gfCNCPoint6[8476] = {X 389.8299, Y 54.3240, Z -8.0000, A 0.000, B 0.000, C 0.000 }
gfCNCPoint6[8477] = {X 390.6035, Y 54.8101, Z -8.0000, A 0.000, B 0.000, C 0.000 }
gfCNCPoint6[8478] = {X 391.2496, Y 55.4562, Z -8.0000, A 0.000, B 0.000, C 0.000 }
gfCNCPoint6[8479] = {X 391.7356, Y 56.2298, Z -8.0000, A 0.000, B 0.000, C 0.000 }
gfCNCPoint6[8480] = {X 392.0374, Y 57.0921, Z -8.0000, A 0.000, B 0.000, C 0.000 }
gfCNCPoint6[8481] = {X 392.1397, Y 58.0000, Z -8.0000, A 0.000, B 0.000, C 0.000 }
gfCNCPoint6[8482] = {X 392.1397, Y 58.9342, Z -8.0000, A 0.000, B 0.000, C 0.000 }
gfCNCPoint6[8483] = {X 392.0387, Y 59.8361, Z -8.0000, A 0.000, B 0.000, C 0.000 }
gfCNCPoint6[8484] = {X 391.7409, Y 60.6934, Z -8.0000, A 0.000, B 0.000, C 0.000 }
gfCNCPoint6[8485] = {X 391.2105, Y 61.5272, Z -8.0000, A 0.000, B 0.000, C 0.000 }
gfCNCPoint6[8486] = {X 390.4961, Y 62.2101, Z -8.0000, A 0.000, B 0.000, C 0.000 }
gfCNCPoint6[8487] = {X 389.6392, Y 62.7024, Z -8.0000, A 0.000, B 0.000, C 0.000 }
gfCNCPoint6[8488] = {X 388.6895, Y 62.9755, Z -8.0000, A 0.000, B 0.000, C 0.000 }
gfCNCPoint6[8489] = {X 388.5563, Y 62.9947, Z -8.0000, A 0.000, B 0.000, C 0.000 }
gfCNCPoint6[8490] = {X 388.4224, Y 63.0095, Z -8.0000, A 0.000, B 0.000, C 0.000 }
gfCNCPoint6[8491] = {X 388.4203, Y 63.1546, Z -8.0000, A 0.000, B 0.000, C 0.000 }
gfCNCPoint6[8492] = {X 388.4183, Y 84.6157, Z -8.0000, A 0.000, B 0.000, C 0.000 }
gfCNCPoint6[8493] = {X 388.3592, Y 86.2534, Z -8.0000, A 0.000, B 0.000, C 0.000 }
gfCNCPoint6[8494] = {X 388.1574, Y 87.8797, Z -8.0000, A 0.000, B 0.000, C 0.000 }
gfCNCPoint6[8495] = {X 387.8145, Y 89.4823, Z -8.0000, A 0.000, B 0.000, C 0.000 }
gfCNCPoint6[8496] = {X 387.2961, Y 91.0293, Z -8.0000, A 0.000, B 0.000, C 0.000 }
gfCNCPoint6[8497] = {X 386.5671, Y 92.4889, Z -8.0000, A 0.000, B 0.000, C 0.000 }
gfCNCPoint6[8498] = {X 385.6417, Y 93.8327, Z -8.0000, A 0.000, B 0.000, C 0.000 }
gfCNCPoint6[8499] = {X 384.5380, Y 95.0343, Z -8.0000, A 0.000, B 0.000, C 0.000 }
gfCNCPoint6[8500] = {X 383.0366, Y 96.3053, Z -8.0000, A 0.000, B 0.000, C 0.000 }
gfCNCPoint6[8501] = {X 381.4074, Y 97.4078, Z -8.0000, A 0.000, B 0.000, C 0.000 }
gfCNCPoint6[8502] = {X 379.6693, Y 98.3292, Z -8.0000, A 0.000, B 0.000, C 0.000 }
gfCNCPoint6[8503] = {X 377.4136, Y 99.2775, Z -8.0000, A 0.000, B 0.000, C 0.000 }
gfCNCPoint6[8504] = {X 375.0960, Y 100.0622, Z -8.0000, A 0.000, B 0.000, C 0.000 }
gfCNCPoint6[8505] = {X 372.7282, Y 100.6793, Z -8.0000, A 0.000, B 0.000, C 0.000 }
gfCNCPoint6[8506] = {X 369.0580, Y 101.3935, Z -8.0000, A 0.000, B 0.000, C 0.000 }
gfCNCPoint6[8507] = {X 365.3582, Y 101.9340, Z -8.0000, A 0.000, B 0.000, C 0.000 }
gfCNCPoint6[8508] = {X 361.6370, Y 102.2996, Z -8.0000, A 0.000, B 0.000, C 0.000 }
gfCNCPoint6[8509] = {X 355.6353, Y 102.6431, Z -8.0000, A 0.000, B 0.000, C 0.000 }
gfCNCPoint6[8510] = {X 349.6255, Y 102.7879, Z -8.0000, A 0.000, B 0.000, C 0.000 }
gfCNCPoint6[8511] = {X 349.6557, Y 106.7878, Z -8.0000, A 0.000, B 0.000, C 0.000 }
gfCNCPoint6[8512] = {X 349.6556, Y 106.7878, Z -8.0000, A 0.000, B 0.000, C 0.000 }
gfCNCPoint6[8513] = {X 349.6249, Y 102.7077, Z -8.0000, A 0.000, B 0.000, C 0.000 }
gfCNCPoint6[8514] = {X 346.2791, Y 102.7021, Z -8.0000, A 0.000, B 0.000, C 0.000 }
gfCNCPoint6[8515] = {X 342.9340, Y 102.6349, Z -8.0000, A 0.000, B 0.000, C 0.000 }
gfCNCPoint6[8516] = {X 342.4013, Y 102.6162, Z -8.0000, A 0.000, B 0.000, C 0.000 }
gfCNCPoint6[8517] = {X 342.2415, Y 102.6136, Z -8.0000, A 0.000, B 0.000, C 0.000 }
gfCNCPoint6[8518] = {X 337.6107, Y 102.4240, Z -8.0000, A 0.000, B 0.000, C 0.000 }
gfCNCPoint6[8519] = {X 332.9916, Y 102.0451, Z -8.0000, A 0.000, B 0.000, C 0.000 }
gfCNCPoint6[8520] = {X 328.3918, Y 101.4774, Z -8.0000, A 0.000, B 0.000, C 0.000 }
gfCNCPoint6[8521] = {X 325.3437, Y 100.9426, Z -8.0000, A 0.000, B 0.000, C 0.000 }
gfCNCPoint6[8522] = {X 322.3384, Y 100.2041, Z -8.0000, A 0.000, B 0.000, C 0.000 }
gfCNCPoint6[8523] = {X 319.3896, Y 99.2654, Z -8.0000, A 0.000, B 0.000, C 0.000 }
gfCNCPoint6[8524] = {X 317.6756, Y 98.5798, Z -8.0000, A 0.000, B 0.000, C 0.000 }
gfCNCPoint6[8525] = {X 316.0258, Y 97.7518, Z -8.0000, A 0.000, B 0.000, C 0.000 }
gfCNCPoint6[8526] = {X 314.4519, Y 96.7872, Z -8.0000, A 0.000, B 0.000, C 0.000 }
gfCNCPoint6[8527] = {X 312.9652, Y 95.6930, Z -8.0000, A 0.000, B 0.000, C 0.000 }
gfCNCPoint6[8528] = {X 311.8398, Y 94.6644, Z -8.0000, A 0.000, B 0.000, C 0.000 }
gfCNCPoint6[8529] = {X 310.8546, Y 93.5009, Z -8.0000, A 0.000, B 0.000, C 0.000 }
gfCNCPoint6[8530] = {X 310.0255, Y 92.2214, Z -8.0000, A 0.000, B 0.000, C 0.000 }
gfCNCPoint6[8531] = {X 309.3660, Y 90.8468, Z -8.0000, A 0.000, B 0.000, C 0.000 }
gfCNCPoint6[8532] = {X 308.8111, Y 89.0438, Z -8.0000, A 0.000, B 0.000, C 0.000 }
gfCNCPoint6[8533] = {X 308.4634, Y 87.1897, Z -8.0000, A 0.000, B 0.000, C 0.000 }
gfCNCPoint6[8534] = {X 308.3276, Y 85.3082, Z -8.0000, A 0.000, B 0.000, C 0.000 }
gfCNCPoint6[8535] = {X 308.3140, Y 84.6159, Z -8.0000, A 0.000, B 0.000, C 0.000 }
gfCNCPoint6[8536] = {X 308.3153, Y 62.9242, Z -8.0000, A 0.000, B 0.000, C 0.000 }
gfCNCPoint6[8537] = {X 307.4730, Y 62.7731, Z -8.0000, A 0.000, B 0.000, C 0.000 }
gfCNCPoint6[8538] = {X 306.6820, Y 62.4463, Z -8.0000, A 0.000, B 0.000, C 0.000 }
gfCNCPoint6[8539] = {X 305.9787, Y 61.9587, Z -8.0000, A 0.000, B 0.000, C 0.000 }
gfCNCPoint6[8540] = {X 305.3952, Y 61.3327, Z -8.0000, A 0.000, B 0.000, C 0.000 }
gfCNCPoint6[8541] = {X 304.9582, Y 60.5969, Z -8.0000, A 0.000, B 0.000, C 0.000 }
gfCNCPoint6[8542] = {X 304.6878, Y 59.7849, Z -8.0000, A 0.000, B 0.000, C 0.000 }
gfCNCPoint6[8543] = {X 304.5962, Y 58.9341, Z -8.0000, A 0.000, B 0.000, C 0.000 }
gfCNCPoint6[8544] = {X 304.5962, Y 58.0000, Z -8.0000, A 0.000, B 0.000, C 0.000 }
gfCNCPoint6[8545] = {X 304.6965, Y 57.1099, Z -8.0000, A 0.000, B 0.000, C 0.000 }
gfCNCPoint6[8546] = {X 304.9923, Y 56.2645, Z -8.0000, A 0.000, B 0.000, C 0.000 }
gfCNCPoint6[8547] = {X 305.4689, Y 55.5060, Z -8.0000, A 0.000, B 0.000, C 0.000 }
gfCNCPoint6[8548] = {X 306.1023, Y 54.8727, Z -8.0000, A 0.000, B 0.000, C 0.000 }
gfCNCPoint6[8549] = {X 306.8607, Y 54.3961, Z -8.0000, A 0.000, B 0.000, C 0.000 }
gfCNCPoint6[8550] = {X 307.7061, Y 54.1003, Z -8.0000, A 0.000, B 0.000, C 0.000 }
gfCNCPoint6[8551] = {X 308.5962, Y 54.0000, Z -8.0000, A 0.000, B 0.000, C 0.000 }
gfCNCPoint6[8552] = {X 324.3107, Y 54.0000, Z -8.0000, A 0.000, B 0.000, C 0.000 }
gfCNCPoint6[8553] = {X 325.2008, Y 54.1003, Z -8.0000, A 0.000, B 0.000, C 0.000 }
gfCNCPoint6[8554] = {X 326.0462, Y 54.3961, Z -8.0000, A 0.000, B 0.000, C 0.000 }
gfCNCPoint6[8555] = {X 326.8046, Y 54.8727, Z -8.0000, A 0.000, B 0.000, C 0.000 }
gfCNCPoint6[8556] = {X 327.4380, Y 55.5060, Z -8.0000, A 0.000, B 0.000, C 0.000 }
gfCNCPoint6[8557] = {X 327.9146, Y 56.2645, Z -8.0000, A 0.000, B 0.000, C 0.000 }
gfCNCPoint6[8558] = {X 328.2104, Y 57.1099, Z -8.0000, A 0.000, B 0.000, C 0.000 }
gfCNCPoint6[8559] = {X 328.3107, Y 58.0000, Z -8.0000, A 0.000, B 0.000, C 0.000 }
gfCNCPoint6[8560] = {X 328.3107, Y 58.9341, Z -8.0000, A 0.000, B 0.000, C 0.000 }
gfCNCPoint6[8561] = {X 328.2156, Y 59.7845, Z -8.0000, A 0.000, B 0.000, C 0.000 }
gfCNCPoint6[8562] = {X 327.9434, Y 60.5958, Z -8.0000, A 0.000, B 0.000, C 0.000 }
gfCNCPoint6[8563] = {X 327.5064, Y 61.3315, Z -8.0000, A 0.000, B 0.000, C 0.000 }
gfCNCPoint6[8564] = {X 326.9240, Y 61.9586, Z -8.0000, A 0.000, B 0.000, C 0.000 }
gfCNCPoint6[8565] = {X 326.2226, Y 62.4488, Z -8.0000, A 0.000, B 0.000, C 0.000 }
gfCNCPoint6[8566] = {X 325.4337, Y 62.7801, Z -8.0000, A 0.000, B 0.000, C 0.000 }
gfCNCPoint6[8567] = {X 324.5926, Y 62.9377, Z -8.0000, A 0.000, B 0.000, C 0.000 }
gfCNCPoint6[8568] = {X 324.5946, Y 83.2313, Z -8.0000, A 0.000, B 0.000, C 0.000 }
gfCNCPoint6[8569] = {X 324.6081, Y 84.6159, Z -8.0000, A 0.000, B 0.000, C 0.000 }
gfCNCPoint6[8570] = {X 324.6916, Y 85.9176, Z -8.0000, A 0.000, B 0.000, C 0.000 }
gfCNCPoint6[8571] = {X 324.9294, Y 87.2002, Z -8.0000, A 0.000, B 0.000, C 0.000 }
gfCNCPoint6[8572] = {X 325.4490, Y 87.7103, Z -8.0000, A 0.000, B 0.000, C 0.000 }
gfCNCPoint6[8573] = {X 326.0776, Y 88.0775, Z -8.0000, A 0.000, B 0.000, C 0.000 }
gfCNCPoint6[8574] = {X 327.8904, Y 88.8015, Z -8.0000, A 0.000, B 0.000, C 0.000 }
gfCNCPoint6[8575] = {X 329.7768, Y 89.3033, Z -8.0000, A 0.000, B 0.000, C 0.000 }
gfCNCPoint6[8576] = {X 332.8789, Y 89.8598, Z -8.0000, A 0.000, B 0.000, C 0.000 }
gfCNCPoint6[8577] = {X 336.0092, Y 90.2262, Z -8.0000, A 0.000, B 0.000, C 0.000 }
gfCNCPoint6[8578] = {X 340.3892, Y 90.5211, Z -8.0000, A 0.000, B 0.000, C 0.000 }
gfCNCPoint6[8579] = {X 344.7764, Y 90.6753, Z -8.0000, A 0.000, B 0.000, C 0.000 }
gfCNCPoint6[8580] = {X 349.1664, Y 90.6886, Z -8.0000, A 0.000, B 0.000, C 0.000 }
gfCNCPoint6[8581] = {X 353.3283, Y 90.6201, Z -8.0000, A 0.000, B 0.000, C 0.000 }
gfCNCPoint6[8582] = {X 357.4851, Y 90.4005, Z -8.0000, A 0.000, B 0.000, C 0.000 }
gfCNCPoint6[8583] = {X 361.6311, Y 90.0301, Z -8.0000, A 0.000, B 0.000, C 0.000 }
gfCNCPoint6[8584] = {X 363.7299, Y 89.7406, Z -8.0000, A 0.000, B 0.000, C 0.000 }
gfCNCPoint6[8585] = {X 365.8095, Y 89.3352, Z -8.0000, A 0.000, B 0.000, C 0.000 }
gfCNCPoint6[8586] = {X 367.8634, Y 88.8152, Z -8.0000, A 0.000, B 0.000, C 0.000 }
gfCNCPoint6[8587] = {X 368.8291, Y 88.4908, Z -8.0000, A 0.000, B 0.000, C 0.000 }
gfCNCPoint6[8588] = {X 369.7521, Y 88.0599, Z -8.0000, A 0.000, B 0.000, C 0.000 }
gfCNCPoint6[8589] = {X 370.6208, Y 87.5278, Z -8.0000, A 0.000, B 0.000, C 0.000 }
gfCNCPoint6[8590] = {X 370.8574, Y 87.2814, Z -8.0000, A 0.000, B 0.000, C 0.000 }
gfCNCPoint6[8591] = {X 370.9793, Y 86.9624, Z -8.0000, A 0.000, B 0.000, C 0.000 }
gfCNCPoint6[8592] = {X 371.1738, Y 85.4011, Z -8.0000, A 0.000, B 0.000, C 0.000 }
gfCNCPoint6[8593] = {X 371.2387, Y 83.8290, Z -8.0000, A 0.000, B 0.000, C 0.000 }
gfCNCPoint6[8594] = {X 371.2376, Y 63.0401, Z -8.0000, A 0.000, B 0.000, C 0.000 }
gfCNCPoint6[8595] = {X 371.2440, Y 62.9246, Z -8.0000, A 0.000, B 0.000, C 0.000 }
gfCNCPoint6[8596] = {X 371.0714, Y 62.9089, Z -8.0000, A 0.000, B 0.000, C 0.000 }
gfCNCPoint6[8597] = {X 370.8996, Y 62.8858, Z -8.0000, A 0.000, B 0.000, C 0.000 }
gfCNCPoint6[8598] = {X 369.9933, Y 62.6315, Z -8.0000, A 0.000, B 0.000, C 0.000 }
gfCNCPoint6[8599] = {X 369.1714, Y 62.1725, Z -8.0000, A 0.000, B 0.000, C 0.000 }
gfCNCPoint6[8600] = {X 368.4796, Y 61.5342, Z -8.0000, A 0.000, B 0.000, C 0.000 }
gfCNCPoint6[8601] = {X 367.9562, Y 60.7518, Z -8.0000, A 0.000, B 0.000, C 0.000 }
gfCNCPoint6[8602] = {X 367.6300, Y 59.8688, Z -8.0000, A 0.000, B 0.000, C 0.000 }
gfCNCPoint6[8603] = {X 367.5193, Y 58.9341, Z -8.0000, A 0.000, B 0.000, C 0.000 }
gfCNCPoint6[8604] = {X 367.5193, Y 58.0000, Z -8.0000, A 0.000, B 0.000, C 0.000 }
gfCNCPoint6[8605] = {X 367.6196, Y 57.1099, Z -8.0000, A 0.000, B 0.000, C 0.000 }
gfCNCPoint6[8606] = {X 367.9154, Y 56.2645, Z -8.0000, A 0.000, B 0.000, C 0.000 }
gfCNCPoint6[8607] = {X 368.3920, Y 55.5060, Z -8.0000, A 0.000, B 0.000, C 0.000 }
gfCNCPoint6[8608] = {X 369.0253, Y 54.8727, Z -8.0000, A 0.000, B 0.000, C 0.000 }
gfCNCPoint6[8609] = {X 369.7837, Y 54.3961, Z -8.0000, A 0.000, B 0.000, C 0.000 }
gfCNCPoint6[8610] = {X 370.6292, Y 54.1003, Z -8.0000, A 0.000, B 0.000, C 0.000 }
gfCNCPoint6[8611] = {X 371.5193, Y 54.0000, Z -8.0000, A 0.000, B 0.000, C 0.000 }
gfCNCPoint6[8612] = {X 388.0597, Y 54.0000, Z -8.0000, A 0.000, B 0.000, C 0.000 }
gfCNCPoint6[8613] = {X 388.9498, Y 54.1003, Z -8.0000, A 0.000, B 0.000, C 0.000 }
gfCNCPoint6[8614] = {X 389.7952, Y 54.3961, Z -8.0000, A 0.000, B 0.000, C 0.000 }
gfCNCPoint6[8615] = {X 390.5536, Y 54.8727, Z -8.0000, A 0.000, B 0.000, C 0.000 }
gfCNCPoint6[8616] = {X 391.1870, Y 55.5060, Z -8.0000, A 0.000, B 0.000, C 0.000 }
gfCNCPoint6[8617] = {X 391.6636, Y 56.2645, Z -8.0000, A 0.000, B 0.000, C 0.000 }
gfCNCPoint6[8618] = {X 391.9594, Y 57.1099, Z -8.0000, A 0.000, B 0.000, C 0.000 }
gfCNCPoint6[8619] = {X 392.0597, Y 58.0000, Z -8.0000, A 0.000, B 0.000, C 0.000 }
gfCNCPoint6[8620] = {X 392.0595, Y 58.9671, Z -8.0000, A 0.000, B 0.000, C 0.000 }
gfCNCPoint6[8621] = {X 391.9570, Y 59.8345, Z -8.0000, A 0.000, B 0.000, C 0.000 }
gfCNCPoint6[8622] = {X 391.6687, Y 60.6589, Z -8.0000, A 0.000, B 0.000, C 0.000 }
gfCNCPoint6[8623] = {X 391.1486, Y 61.4765, Z -8.0000, A 0.000, B 0.000, C 0.000 }
gfCNCPoint6[8624] = {X 390.4482, Y 62.1460, Z -8.0000, A 0.000, B 0.000, C 0.000 }
gfCNCPoint6[8625] = {X 389.6080, Y 62.6287, Z -8.0000, A 0.000, B 0.000, C 0.000 }
gfCNCPoint6[8626] = {X 388.6768, Y 62.8965, Z -8.0000, A 0.000, B 0.000, C 0.000 }
gfCNCPoint6[8627] = {X 388.5106, Y 62.9197, Z -8.0000, A 0.000, B 0.000, C 0.000 }
gfCNCPoint6[8628] = {X 388.3435, Y 62.9359, Z -8.0000, A 0.000, B 0.000, C 0.000 }
gfCNCPoint6[8629] = {X 388.3403, Y 63.1540, Z -8.0000, A 0.000, B 0.000, C 0.000 }
gfCNCPoint6[8630] = {X 388.3403, Y 83.9236, Z -8.0000, A 0.000, B 0.000, C 0.000 }
gfCNCPoint6[8631] = {X 388.3383, Y 84.6159, Z -8.0000, A 0.000, B 0.000, C 0.000 }
gfCNCPoint6[8632] = {X 388.2794, Y 86.2468, Z -8.0000, A 0.000, B 0.000, C 0.000 }
gfCNCPoint6[8633] = {X 388.0785, Y 87.8663, Z -8.0000, A 0.000, B 0.000, C 0.000 }
gfCNCPoint6[8634] = {X 387.7371, Y 89.4621, Z -8.0000, A 0.000, B 0.000, C 0.000 }
gfCNCPoint6[8635] = {X 387.2222, Y 90.9986, Z -8.0000, A 0.000, B 0.000, C 0.000 }
gfCNCPoint6[8636] = {X 386.4982, Y 92.4482, Z -8.0000, A 0.000, B 0.000, C 0.000 }
gfCNCPoint6[8637] = {X 385.5792, Y 93.7828, Z -8.0000, A 0.000, B 0.000, C 0.000 }
gfCNCPoint6[8638] = {X 384.4830, Y 94.9762, Z -8.0000, A 0.000, B 0.000, C 0.000 }
gfCNCPoint6[8639] = {X 382.9881, Y 96.2416, Z -8.0000, A 0.000, B 0.000, C 0.000 }
gfCNCPoint6[8640] = {X 381.3661, Y 97.3393, Z -8.0000, A 0.000, B 0.000, C 0.000 }
gfCNCPoint6[8641] = {X 379.6357, Y 98.2566, Z -8.0000, A 0.000, B 0.000, C 0.000 }
gfCNCPoint6[8642] = {X 377.3853, Y 99.2027, Z -8.0000, A 0.000, B 0.000, C 0.000 }
gfCNCPoint6[8643] = {X 375.0731, Y 99.9856, Z -8.0000, A 0.000, B 0.000, C 0.000 }
gfCNCPoint6[8644] = {X 372.7108, Y 100.6012, Z -8.0000, A 0.000, B 0.000, C 0.000 }
gfCNCPoint6[8645] = {X 369.0444, Y 101.3146, Z -8.0000, A 0.000, B 0.000, C 0.000 }
gfCNCPoint6[8646] = {X 365.3484, Y 101.8546, Z -8.0000, A 0.000, B 0.000, C 0.000 }
gfCNCPoint6[8647] = {X 361.6311, Y 102.2198, Z -8.0000, A 0.000, B 0.000, C 0.000 }
gfCNCPoint6[8648] = {X 355.6320, Y 102.5630, Z -8.0000, A 0.000, B 0.000, C 0.000 }
gfCNCPoint6[8649] = {X 349.6249, Y 102.7077, Z -8.0000, A 0.000, B 0.000, C 0.000 }
gfCNCPoint6[8650] = {X 349.6556, Y 106.7878, Z -8.0000, A 0.000, B 0.000, C 0.000 }
gfCNCPoint6[8651] = {X 349.6556, Y 106.7878, Z -5.0000, A 0.000, B 0.000, C 0.000 }
gfCNCPoint6[8652] = {X 349.6556, Y 106.7878, Z 11.0000, A 0.000, B 0.000, C 0.000 }
gfCNCPoint6[8653] = {X 411.5981, Y 79.5921, Z 11.0000, A 0.000, B 0.000, C 0.000 }
gfCNCPoint6[8654] = {X 411.5981, Y 79.5921, Z -5.0000, A 0.000, B 0.000, C 0.000 }
gfCNCPoint6[8655] = {X 411.5981, Y 79.5921, Z -8.0000, A 0.000, B 0.000, C 0.000 }
gfCNCPoint6[8656] = {X 413.7984, Y 83.0280, Z -8.0000, A 0.000, B 0.000, C 0.000 }
gfCNCPoint6[8657] = {X 428.0532, Y 73.8997, Z -8.0000, A 0.000, B 0.000, C 0.000 }
gfCNCPoint6[8658] = {X 403.7556, Y 64.3672, Z -8.0000, A 0.000, B 0.000, C 0.000 }
gfCNCPoint6[8659] = {X 402.0595, Y 63.8058, Z -8.0000, A 0.000, B 0.000, C 0.000 }
gfCNCPoint6[8660] = {X 400.3122, Y 63.4333, Z -8.0000, A 0.000, B 0.000, C 0.000 }
gfCNCPoint6[8661] = {X 398.5347, Y 63.2540, Z -8.0000, A 0.000, B 0.000, C 0.000 }
gfCNCPoint6[8662] = {X 397.5821, Y 63.1425, Z -8.0000, A 0.000, B 0.000, C 0.000 }
gfCNCPoint6[8663] = {X 396.6777, Y 62.8235, Z -8.0000, A 0.000, B 0.000, C 0.000 }
gfCNCPoint6[8664] = {X 395.8659, Y 62.3129, Z -8.0000, A 0.000, B 0.000, C 0.000 }
gfCNCPoint6[8665] = {X 395.1868, Y 61.6357, Z -8.0000, A 0.000, B 0.000, C 0.000 }
gfCNCPoint6[8666] = {X 394.6738, Y 60.8255, Z -8.0000, A 0.000, B 0.000, C 0.000 }
gfCNCPoint6[8667] = {X 394.3522, Y 59.9219, Z -8.0000, A 0.000, B 0.000, C 0.000 }
gfCNCPoint6[8668] = {X 394.2379, Y 58.9697, Z -8.0000, A 0.000, B 0.000, C 0.000 }
gfCNCPoint6[8669] = {X 394.2377, Y 58.0000, Z -8.0000, A 0.000, B 0.000, C 0.000 }
gfCNCPoint6[8670] = {X 394.3460, Y 57.0387, Z -8.0000, A 0.000, B 0.000, C 0.000 }
gfCNCPoint6[8671] = {X 394.6655, Y 56.1256, Z -8.0000, A 0.000, B 0.000, C 0.000 }
gfCNCPoint6[8672] = {X 395.1802, Y 55.3065, Z -8.0000, A 0.000, B 0.000, C 0.000 }
gfCNCPoint6[8673] = {X 395.8642, Y 54.6225, Z -8.0000, A 0.000, B 0.000, C 0.000 }
gfCNCPoint6[8674] = {X 396.6833, Y 54.1078, Z -8.0000, A 0.000, B 0.000, C 0.000 }
gfCNCPoint6[8675] = {X 397.5964, Y 53.7883, Z -8.0000, A 0.000, B 0.000, C 0.000 }
gfCNCPoint6[8676] = {X 398.5577, Y 53.6800, Z -8.0000, A 0.000, B 0.000, C 0.000 }
gfCNCPoint6[8677] = {X 419.4886, Y 53.6800, Z -8.0000, A 0.000, B 0.000, C 0.000 }
gfCNCPoint6[8678] = {X 420.4499, Y 53.7883, Z -8.0000, A 0.000, B 0.000, C 0.000 }
gfCNCPoint6[8679] = {X 421.3630, Y 54.1078, Z -8.0000, A 0.000, B 0.000, C 0.000 }
gfCNCPoint6[8680] = {X 422.1821, Y 54.6225, Z -8.0000, A 0.000, B 0.000, C 0.000 }
gfCNCPoint6[8681] = {X 422.8661, Y 55.3065, Z -8.0000, A 0.000, B 0.000, C 0.000 }
gfCNCPoint6[8682] = {X 423.3808, Y 56.1256, Z -8.0000, A 0.000, B 0.000, C 0.000 }
gfCNCPoint6[8683] = {X 423.7003, Y 57.0387, Z -8.0000, A 0.000, B 0.000, C 0.000 }
gfCNCPoint6[8684] = {X 423.8086, Y 58.0000, Z -8.0000, A 0.000, B 0.000, C 0.000 }
gfCNCPoint6[8685] = {X 423.8086, Y 58.2314, Z -8.0000, A 0.000, B 0.000, C 0.000 }
gfCNCPoint6[8686] = {X 429.6116, Y 60.4920, Z -8.0000, A 0.000, B 0.000, C 0.000 }
gfCNCPoint6[8687] = {X 457.8579, Y 71.6995, Z -8.0000, A 0.000, B 0.000, C 0.000 }
gfCNCPoint6[8688] = {X 457.8601, Y 63.2123, Z -8.0000, A 0.000, B 0.000, C 0.000 }
gfCNCPoint6[8689] = {X 457.0085, Y 63.0031, Z -8.0000, A 0.000, B 0.000, C 0.000 }
gfCNCPoint6[8690] = {X 456.2167, Y 62.6262, Z -8.0000, A 0.000, B 0.000, C 0.000 }
gfCNCPoint6[8691] = {X 455.5174, Y 62.0973, Z -8.0000, A 0.000, B 0.000, C 0.000 }
gfCNCPoint6[8692] = {X 454.9393, Y 61.4380, Z -8.0000, A 0.000, B 0.000, C 0.000 }
gfCNCPoint6[8693] = {X 454.5062, Y 60.6755, Z -8.0000, A 0.000, B 0.000, C 0.000 }
gfCNCPoint6[8694] = {X 454.2359, Y 59.8413, Z -8.0000, A 0.000, B 0.000, C 0.000 }
gfCNCPoint6[8695] = {X 454.1398, Y 58.9697, Z -8.0000, A 0.000, B 0.000, C 0.000 }
gfCNCPoint6[8696] = {X 454.1396, Y 58.0000, Z -8.0000, A 0.000, B 0.000, C 0.000 }
gfCNCPoint6[8697] = {X 454.2479, Y 57.0387, Z -8.0000, A 0.000, B 0.000, C 0.000 }
gfCNCPoint6[8698] = {X 454.5674, Y 56.1256, Z -8.0000, A 0.000, B 0.000, C 0.000 }
gfCNCPoint6[8699] = {X 455.0821, Y 55.3065, Z -8.0000, A 0.000, B 0.000, C 0.000 }
gfCNCPoint6[8700] = {X 455.7661, Y 54.6225, Z -8.0000, A 0.000, B 0.000, C 0.000 }
gfCNCPoint6[8701] = {X 456.5852, Y 54.1078, Z -8.0000, A 0.000, B 0.000, C 0.000 }
gfCNCPoint6[8702] = {X 457.4983, Y 53.7883, Z -8.0000, A 0.000, B 0.000, C 0.000 }
gfCNCPoint6[8703] = {X 458.4596, Y 53.6800, Z -8.0000, A 0.000, B 0.000, C 0.000 }
gfCNCPoint6[8704] = {X 475.0000, Y 53.6800, Z -8.0000, A 0.000, B 0.000, C 0.000 }
gfCNCPoint6[8705] = {X 475.9613, Y 53.7883, Z -8.0000, A 0.000, B 0.000, C 0.000 }
gfCNCPoint6[8706] = {X 476.8744, Y 54.1078, Z -8.0000, A 0.000, B 0.000, C 0.000 }
gfCNCPoint6[8707] = {X 477.6935, Y 54.6225, Z -8.0000, A 0.000, B 0.000, C 0.000 }
gfCNCPoint6[8708] = {X 478.3775, Y 55.3065, Z -8.0000, A 0.000, B 0.000, C 0.000 }
gfCNCPoint6[8709] = {X 478.8922, Y 56.1256, Z -8.0000, A 0.000, B 0.000, C 0.000 }
gfCNCPoint6[8710] = {X 479.2117, Y 57.0387, Z -8.0000, A 0.000, B 0.000, C 0.000 }
gfCNCPoint6[8711] = {X 479.3200, Y 58.0000, Z -8.0000, A 0.000, B 0.000, C 0.000 }
gfCNCPoint6[8712] = {X 479.3200, Y 58.9342, Z -8.0000, A 0.000, B 0.000, C 0.000 }
gfCNCPoint6[8713] = {X 479.2300, Y 59.8113, Z -8.0000, A 0.000, B 0.000, C 0.000 }
gfCNCPoint6[8714] = {X 478.9638, Y 60.6518, Z -8.0000, A 0.000, B 0.000, C 0.000 }
gfCNCPoint6[8715] = {X 478.5325, Y 61.4208, Z -8.0000, A 0.000, B 0.000, C 0.000 }
gfCNCPoint6[8716] = {X 477.9541, Y 62.0862, Z -8.0000, A 0.000, B 0.000, C 0.000 }
gfCNCPoint6[8717] = {X 477.2526, Y 62.6203, Z -8.0000, A 0.000, B 0.000, C 0.000 }
gfCNCPoint6[8718] = {X 476.4572, Y 63.0009, Z -8.0000, A 0.000, B 0.000, C 0.000 }
gfCNCPoint6[8719] = {X 475.6012, Y 63.2120, Z -8.0000, A 0.000, B 0.000, C 0.000 }
gfCNCPoint6[8720] = {X 475.6017, Y 92.7672, Z -8.0000, A 0.000, B 0.000, C 0.000 }
gfCNCPoint6[8721] = {X 475.9938, Y 92.8650, Z -8.0000, A 0.000, B 0.000, C 0.000 }
gfCNCPoint6[8722] = {X 476.3804, Y 92.9828, Z -8.0000, A 0.000, B 0.000, C 0.000 }
gfCNCPoint6[8723] = {X 477.1940, Y 93.3517, Z -8.0000, A 0.000, B 0.000, C 0.000 }
gfCNCPoint6[8724] = {X 477.9137, Y 93.8808, Z -8.0000, A 0.000, B 0.000, C 0.000 }
gfCNCPoint6[8725] = {X 478.5085, Y 94.5472, Z -8.0000, A 0.000, B 0.000, C 0.000 }
gfCNCPoint6[8726] = {X 478.9527, Y 95.3222, Z -8.0000, A 0.000, B 0.000, C 0.000 }
gfCNCPoint6[8727] = {X 479.2272, Y 96.1722, Z -8.0000, A 0.000, B 0.000, C 0.000 }
gfCNCPoint6[8728] = {X 479.3200, Y 97.0606, Z -8.0000, A 0.000, B 0.000, C 0.000 }
gfCNCPoint6[8729] = {X 479.3200, Y 98.0000, Z -8.0000, A 0.000, B 0.000, C 0.000 }
gfCNCPoint6[8730] = {X 479.2117, Y 98.9613, Z -8.0000, A 0.000, B 0.000, C 0.000 }
gfCNCPoint6[8731] = {X 478.8922, Y 99.8744, Z -8.0000, A 0.000, B 0.000, C 0.000 }
gfCNCPoint6[8732] = {X 478.3775, Y 100.6935, Z -8.0000, A 0.000, B 0.000, C 0.000 }
gfCNCPoint6[8733] = {X 477.6935, Y 101.3775, Z -8.0000, A 0.000, B 0.000, C 0.000 }
gfCNCPoint6[8734] = {X 476.8744, Y 101.8922, Z -8.0000, A 0.000, B 0.000, C 0.000 }
gfCNCPoint6[8735] = {X 475.9613, Y 102.2117, Z -8.0000, A 0.000, B 0.000, C 0.000 }
gfCNCPoint6[8736] = {X 475.0000, Y 102.3200, Z -8.0000, A 0.000, B 0.000, C 0.000 }
gfCNCPoint6[8737] = {X 458.4596, Y 102.3200, Z -8.0000, A 0.000, B 0.000, C 0.000 }
gfCNCPoint6[8738] = {X 457.4983, Y 102.2117, Z -8.0000, A 0.000, B 0.000, C 0.000 }
gfCNCPoint6[8739] = {X 456.5852, Y 101.8922, Z -8.0000, A 0.000, B 0.000, C 0.000 }
gfCNCPoint6[8740] = {X 455.7661, Y 101.3775, Z -8.0000, A 0.000, B 0.000, C 0.000 }
gfCNCPoint6[8741] = {X 455.0821, Y 100.6935, Z -8.0000, A 0.000, B 0.000, C 0.000 }
gfCNCPoint6[8742] = {X 454.5674, Y 99.8744, Z -8.0000, A 0.000, B 0.000, C 0.000 }
gfCNCPoint6[8743] = {X 454.2479, Y 98.9613, Z -8.0000, A 0.000, B 0.000, C 0.000 }
gfCNCPoint6[8744] = {X 454.1396, Y 98.0000, Z -8.0000, A 0.000, B 0.000, C 0.000 }
gfCNCPoint6[8745] = {X 454.1396, Y 97.0659, Z -8.0000, A 0.000, B 0.000, C 0.000 }
gfCNCPoint6[8746] = {X 454.2295, Y 96.1891, Z -8.0000, A 0.000, B 0.000, C 0.000 }
gfCNCPoint6[8747] = {X 454.4955, Y 95.3488, Z -8.0000, A 0.000, B 0.000, C 0.000 }
gfCNCPoint6[8748] = {X 454.9265, Y 94.5800, Z -8.0000, A 0.000, B 0.000, C 0.000 }
gfCNCPoint6[8749] = {X 455.5046, Y 93.9147, Z -8.0000, A 0.000, B 0.000, C 0.000 }
gfCNCPoint6[8750] = {X 456.2057, Y 93.3805, Z -8.0000, A 0.000, B 0.000, C 0.000 }
gfCNCPoint6[8751] = {X 457.0006, Y 92.9998, Z -8.0000, A 0.000, B 0.000, C 0.000 }
gfCNCPoint6[8752] = {X 457.8563, Y 92.7883, Z -8.0000, A 0.000, B 0.000, C 0.000 }
gfCNCPoint6[8753] = {X 457.8563, Y 85.5950, Z -8.0000, A 0.000, B 0.000, C 0.000 }
gfCNCPoint6[8754] = {X 444.8604, Y 80.5006, Z -8.0000, A 0.000, B 0.000, C 0.000 }
gfCNCPoint6[8755] = {X 420.0244, Y 96.5885, Z -8.0000, A 0.000, B 0.000, C 0.000 }
gfCNCPoint6[8756] = {X 420.0267, Y 97.0651, Z -8.0000, A 0.000, B 0.000, C 0.000 }
gfCNCPoint6[8757] = {X 420.0267, Y 98.0000, Z -8.0000, A 0.000, B 0.000, C 0.000 }
gfCNCPoint6[8758] = {X 419.9184, Y 98.9613, Z -8.0000, A 0.000, B 0.000, C 0.000 }
gfCNCPoint6[8759] = {X 419.5989, Y 99.8744, Z -8.0000, A 0.000, B 0.000, C 0.000 }
gfCNCPoint6[8760] = {X 419.0842, Y 100.6935, Z -8.0000, A 0.000, B 0.000, C 0.000 }
gfCNCPoint6[8761] = {X 418.4002, Y 101.3775, Z -8.0000, A 0.000, B 0.000, C 0.000 }
gfCNCPoint6[8762] = {X 417.5811, Y 101.8922, Z -8.0000, A 0.000, B 0.000, C 0.000 }
gfCNCPoint6[8763] = {X 416.6680, Y 102.2117, Z -8.0000, A 0.000, B 0.000, C 0.000 }
gfCNCPoint6[8764] = {X 415.7067, Y 102.3200, Z -8.0000, A 0.000, B 0.000, C 0.000 }
gfCNCPoint6[8765] = {X 396.4059, Y 102.3200, Z -8.0000, A 0.000, B 0.000, C 0.000 }
gfCNCPoint6[8766] = {X 395.4447, Y 102.2117, Z -8.0000, A 0.000, B 0.000, C 0.000 }
gfCNCPoint6[8767] = {X 394.5316, Y 101.8922, Z -8.0000, A 0.000, B 0.000, C 0.000 }
gfCNCPoint6[8768] = {X 393.7125, Y 101.3775, Z -8.0000, A 0.000, B 0.000, C 0.000 }
gfCNCPoint6[8769] = {X 393.0284, Y 100.6935, Z -8.0000, A 0.000, B 0.000, C 0.000 }
gfCNCPoint6[8770] = {X 392.5138, Y 99.8744, Z -8.0000, A 0.000, B 0.000, C 0.000 }
gfCNCPoint6[8771] = {X 392.1943, Y 98.9613, Z -8.0000, A 0.000, B 0.000, C 0.000 }
gfCNCPoint6[8772] = {X 392.0859, Y 98.0000, Z -8.0000, A 0.000, B 0.000, C 0.000 }
gfCNCPoint6[8773] = {X 392.0859, Y 97.0659, Z -8.0000, A 0.000, B 0.000, C 0.000 }
gfCNCPoint6[8774] = {X 392.1937, Y 96.1069, Z -8.0000, A 0.000, B 0.000, C 0.000 }
gfCNCPoint6[8775] = {X 392.5117, Y 95.1958, Z -8.0000, A 0.000, B 0.000, C 0.000 }
gfCNCPoint6[8776] = {X 393.0240, Y 94.3780, Z -8.0000, A 0.000, B 0.000, C 0.000 }
gfCNCPoint6[8777] = {X 393.7051, Y 93.6943, Z -8.0000, A 0.000, B 0.000, C 0.000 }
gfCNCPoint6[8778] = {X 394.5210, Y 93.1789, Z -8.0000, A 0.000, B 0.000, C 0.000 }
gfCNCPoint6[8779] = {X 395.4309, Y 92.8574, Z -8.0000, A 0.000, B 0.000, C 0.000 }
gfCNCPoint6[8780] = {X 396.3894, Y 92.7460, Z -8.0000, A 0.000, B 0.000, C 0.000 }
gfCNCPoint6[8781] = {X 397.3432, Y 92.7029, Z -8.0000, A 0.000, B 0.000, C 0.000 }
gfCNCPoint6[8782] = {X 398.2936, Y 92.6130, Z -8.0000, A 0.000, B 0.000, C 0.000 }
gfCNCPoint6[8783] = {X 398.9444, Y 92.4553, Z -8.0000, A 0.000, B 0.000, C 0.000 }
gfCNCPoint6[8784] = {X 399.5436, Y 92.1563, Z -8.0000, A 0.000, B 0.000, C 0.000 }
gfCNCPoint6[8785] = {X 413.7984, Y 83.0280, Z -8.0000, A 0.000, B 0.000, C 0.000 }
gfCNCPoint6[8786] = {X 411.6413, Y 79.6595, Z -8.0000, A 0.000, B 0.000, C 0.000 }
gfCNCPoint6[8787] = {X 413.8415, Y 83.0954, Z -8.0000, A 0.000, B 0.000, C 0.000 }
gfCNCPoint6[8788] = {X 428.2284, Y 73.8825, Z -8.0000, A 0.000, B 0.000, C 0.000 }
gfCNCPoint6[8789] = {X 403.7848, Y 64.2927, Z -8.0000, A 0.000, B 0.000, C 0.000 }
gfCNCPoint6[8790] = {X 402.0799, Y 63.7285, Z -8.0000, A 0.000, B 0.000, C 0.000 }
gfCNCPoint6[8791] = {X 400.3235, Y 63.3541, Z -8.0000, A 0.000, B 0.000, C 0.000 }
gfCNCPoint6[8792] = {X 398.5367, Y 63.1740, Z -8.0000, A 0.000, B 0.000, C 0.000 }
gfCNCPoint6[8793] = {X 397.6016, Y 63.0648, Z -8.0000, A 0.000, B 0.000, C 0.000 }
gfCNCPoint6[8794] = {X 396.7136, Y 62.7520, Z -8.0000, A 0.000, B 0.000, C 0.000 }
gfCNCPoint6[8795] = {X 395.9165, Y 62.2509, Z -8.0000, A 0.000, B 0.000, C 0.000 }
gfCNCPoint6[8796] = {X 395.2496, Y 61.5863, Z -8.0000, A 0.000, B 0.000, C 0.000 }
gfCNCPoint6[8797] = {X 394.7459, Y 60.7908, Z -8.0000, A 0.000, B 0.000, C 0.000 }
gfCNCPoint6[8798] = {X 394.4301, Y 59.9039, Z -8.0000, A 0.000, B 0.000, C 0.000 }
gfCNCPoint6[8799] = {X 394.3179, Y 58.9691, Z -8.0000, A 0.000, B 0.000, C 0.000 }
gfCNCPoint6[8800] = {X 394.3177, Y 58.0000, Z -8.0000, A 0.000, B 0.000, C 0.000 }
gfCNCPoint6[8801] = {X 394.4240, Y 57.0565, Z -8.0000, A 0.000, B 0.000, C 0.000 }
gfCNCPoint6[8802] = {X 394.7376, Y 56.1603, Z -8.0000, A 0.000, B 0.000, C 0.000 }
gfCNCPoint6[8803] = {X 395.2428, Y 55.3564, Z -8.0000, A 0.000, B 0.000, C 0.000 }
gfCNCPoint6[8804] = {X 395.9141, Y 54.6850, Z -8.0000, A 0.000, B 0.000, C 0.000 }
gfCNCPoint6[8805] = {X 396.7181, Y 54.1799, Z -8.0000, A 0.000, B 0.000, C 0.000 }
gfCNCPoint6[8806] = {X 397.6142, Y 53.8663, Z -8.0000, A 0.000, B 0.000, C 0.000 }
gfCNCPoint6[8807] = {X 398.5577, Y 53.7600, Z -8.0000, A 0.000, B 0.000, C 0.000 }
gfCNCPoint6[8808] = {X 419.4886, Y 53.7600, Z -8.0000, A 0.000, B 0.000, C 0.000 }
gfCNCPoint6[8809] = {X 420.4321, Y 53.8663, Z -8.0000, A 0.000, B 0.000, C 0.000 }
gfCNCPoint6[8810] = {X 421.3283, Y 54.1799, Z -8.0000, A 0.000, B 0.000, C 0.000 }
gfCNCPoint6[8811] = {X 422.1322, Y 54.6850, Z -8.0000, A 0.000, B 0.000, C 0.000 }
gfCNCPoint6[8812] = {X 422.8036, Y 55.3564, Z -8.0000, A 0.000, B 0.000, C 0.000 }
gfCNCPoint6[8813] = {X 423.3087, Y 56.1603, Z -8.0000, A 0.000, B 0.000, C 0.000 }
gfCNCPoint6[8814] = {X 423.6223, Y 57.0565, Z -8.0000, A 0.000, B 0.000, C 0.000 }
gfCNCPoint6[8815] = {X 423.7286, Y 58.0000, Z -8.0000, A 0.000, B 0.000, C 0.000 }
gfCNCPoint6[8816] = {X 423.7286, Y 58.2861, Z -8.0000, A 0.000, B 0.000, C 0.000 }
gfCNCPoint6[8817] = {X 429.5823, Y 60.5665, Z -8.0000, A 0.000, B 0.000, C 0.000 }
gfCNCPoint6[8818] = {X 457.9378, Y 71.8173, Z -8.0000, A 0.000, B 0.000, C 0.000 }
gfCNCPoint6[8819] = {X 457.9401, Y 63.1421, Z -8.0000, A 0.000, B 0.000, C 0.000 }
gfCNCPoint6[8820] = {X 457.0916, Y 62.9473, Z -8.0000, A 0.000, B 0.000, C 0.000 }
gfCNCPoint6[8821] = {X 456.3009, Y 62.5834, Z -8.0000, A 0.000, B 0.000, C 0.000 }
gfCNCPoint6[8822] = {X 455.6011, Y 62.0656, Z -8.0000, A 0.000, B 0.000, C 0.000 }
gfCNCPoint6[8823] = {X 455.0218, Y 61.4158, Z -8.0000, A 0.000, B 0.000, C 0.000 }
gfCNCPoint6[8824] = {X 454.5874, Y 60.6614, Z -8.0000, A 0.000, B 0.000, C 0.000 }
gfCNCPoint6[8825] = {X 454.3163, Y 59.8342, Z -8.0000, A 0.000, B 0.000, C 0.000 }
gfCNCPoint6[8826] = {X 454.2197, Y 58.9691, Z -8.0000, A 0.000, B 0.000, C 0.000 }
gfCNCPoint6[8827] = {X 454.2196, Y 58.0000, Z -8.0000, A 0.000, B 0.000, C 0.000 }
gfCNCPoint6[8828] = {X 454.3259, Y 57.0565, Z -8.0000, A 0.000, B 0.000, C 0.000 }
gfCNCPoint6[8829] = {X 454.6395, Y 56.1603, Z -8.0000, A 0.000, B 0.000, C 0.000 }
gfCNCPoint6[8830] = {X 455.1446, Y 55.3564, Z -8.0000, A 0.000, B 0.000, C 0.000 }
gfCNCPoint6[8831] = {X 455.8160, Y 54.6850, Z -8.0000, A 0.000, B 0.000, C 0.000 }
gfCNCPoint6[8832] = {X 456.6199, Y 54.1799, Z -8.0000, A 0.000, B 0.000, C 0.000 }
gfCNCPoint6[8833] = {X 457.5161, Y 53.8663, Z -8.0000, A 0.000, B 0.000, C 0.000 }
gfCNCPoint6[8834] = {X 458.4596, Y 53.7600, Z -8.0000, A 0.000, B 0.000, C 0.000 }
gfCNCPoint6[8835] = {X 475.0000, Y 53.7600, Z -8.0000, A 0.000, B 0.000, C 0.000 }
gfCNCPoint6[8836] = {X 475.9435, Y 53.8663, Z -8.0000, A 0.000, B 0.000, C 0.000 }
gfCNCPoint6[8837] = {X 476.8397, Y 54.1799, Z -8.0000, A 0.000, B 0.000, C 0.000 }
gfCNCPoint6[8838] = {X 477.6436, Y 54.6850, Z -8.0000, A 0.000, B 0.000, C 0.000 }
gfCNCPoint6[8839] = {X 478.3150, Y 55.3564, Z -8.0000, A 0.000, B 0.000, C 0.000 }
gfCNCPoint6[8840] = {X 478.8201, Y 56.1603, Z -8.0000, A 0.000, B 0.000, C 0.000 }
gfCNCPoint6[8841] = {X 479.1337, Y 57.0565, Z -8.0000, A 0.000, B 0.000, C 0.000 }
gfCNCPoint6[8842] = {X 479.2400, Y 58.0000, Z -8.0000, A 0.000, B 0.000, C 0.000 }
gfCNCPoint6[8843] = {X 479.2400, Y 58.9342, Z -8.0000, A 0.000, B 0.000, C 0.000 }
gfCNCPoint6[8844] = {X 479.1496, Y 59.8048, Z -8.0000, A 0.000, B 0.000, C 0.000 }
gfCNCPoint6[8845] = {X 478.8825, Y 60.6382, Z -8.0000, A 0.000, B 0.000, C 0.000 }
gfCNCPoint6[8846] = {X 478.4499, Y 61.3990, Z -8.0000, A 0.000, B 0.000, C 0.000 }
gfCNCPoint6[8847] = {X 477.8703, Y 62.0548, Z -8.0000, A 0.000, B 0.000, C 0.000 }
gfCNCPoint6[8848] = {X 477.1684, Y 62.5777, Z -8.0000, A 0.000, B 0.000, C 0.000 }
gfCNCPoint6[8849] = {X 476.3741, Y 62.9452, Z -8.0000, A 0.000, B 0.000, C 0.000 }
gfCNCPoint6[8850] = {X 475.5212, Y 63.1419, Z -8.0000, A 0.000, B 0.000, C 0.000 }
gfCNCPoint6[8851] = {X 475.5217, Y 92.8316, Z -8.0000, A 0.000, B 0.000, C 0.000 }
gfCNCPoint6[8852] = {X 475.9416, Y 92.9336, Z -8.0000, A 0.000, B 0.000, C 0.000 }
gfCNCPoint6[8853] = {X 476.3551, Y 93.0587, Z -8.0000, A 0.000, B 0.000, C 0.000 }
gfCNCPoint6[8854] = {X 477.1535, Y 93.4207, Z -8.0000, A 0.000, B 0.000, C 0.000 }
gfCNCPoint6[8855] = {X 477.8599, Y 93.9400, Z -8.0000, A 0.000, B 0.000, C 0.000 }
gfCNCPoint6[8856] = {X 478.4436, Y 94.5940, Z -8.0000, A 0.000, B 0.000, C 0.000 }
gfCNCPoint6[8857] = {X 478.8796, Y 95.3545, Z -8.0000, A 0.000, B 0.000, C 0.000 }
gfCNCPoint6[8858] = {X 479.1489, Y 96.1887, Z -8.0000, A 0.000, B 0.000, C 0.000 }
gfCNCPoint6[8859] = {X 479.2400, Y 97.0606, Z -8.0000, A 0.000, B 0.000, C 0.000 }
gfCNCPoint6[8860] = {X 479.2400, Y 98.0000, Z -8.0000, A 0.000, B 0.000, C 0.000 }
gfCNCPoint6[8861] = {X 479.1337, Y 98.9435, Z -8.0000, A 0.000, B 0.000, C 0.000 }
gfCNCPoint6[8862] = {X 478.8201, Y 99.8397, Z -8.0000, A 0.000, B 0.000, C 0.000 }
gfCNCPoint6[8863] = {X 478.3150, Y 100.6436, Z -8.0000, A 0.000, B 0.000, C 0.000 }
gfCNCPoint6[8864] = {X 477.6436, Y 101.3150, Z -8.0000, A 0.000, B 0.000, C 0.000 }
gfCNCPoint6[8865] = {X 476.8397, Y 101.8201, Z -8.0000, A 0.000, B 0.000, C 0.000 }
gfCNCPoint6[8866] = {X 475.9435, Y 102.1337, Z -8.0000, A 0.000, B 0.000, C 0.000 }
gfCNCPoint6[8867] = {X 475.0000, Y 102.2400, Z -8.0000, A 0.000, B 0.000, C 0.000 }
gfCNCPoint6[8868] = {X 458.4596, Y 102.2400, Z -8.0000, A 0.000, B 0.000, C 0.000 }
gfCNCPoint6[8869] = {X 457.5161, Y 102.1337, Z -8.0000, A 0.000, B 0.000, C 0.000 }
gfCNCPoint6[8870] = {X 456.6199, Y 101.8201, Z -8.0000, A 0.000, B 0.000, C 0.000 }
gfCNCPoint6[8871] = {X 455.8160, Y 101.3150, Z -8.0000, A 0.000, B 0.000, C 0.000 }
gfCNCPoint6[8872] = {X 455.1446, Y 100.6436, Z -8.0000, A 0.000, B 0.000, C 0.000 }
gfCNCPoint6[8873] = {X 454.6395, Y 99.8397, Z -8.0000, A 0.000, B 0.000, C 0.000 }
gfCNCPoint6[8874] = {X 454.3259, Y 98.9435, Z -8.0000, A 0.000, B 0.000, C 0.000 }
gfCNCPoint6[8875] = {X 454.2196, Y 98.0000, Z -8.0000, A 0.000, B 0.000, C 0.000 }
gfCNCPoint6[8876] = {X 454.2196, Y 97.0659, Z -8.0000, A 0.000, B 0.000, C 0.000 }
gfCNCPoint6[8877] = {X 454.3099, Y 96.1957, Z -8.0000, A 0.000, B 0.000, C 0.000 }
gfCNCPoint6[8878] = {X 454.5769, Y 95.3624, Z -8.0000, A 0.000, B 0.000, C 0.000 }
gfCNCPoint6[8879] = {X 455.0092, Y 94.6018, Z -8.0000, A 0.000, B 0.000, C 0.000 }
gfCNCPoint6[8880] = {X 455.5884, Y 93.9460, Z -8.0000, A 0.000, B 0.000, C 0.000 }
gfCNCPoint6[8881] = {X 456.2899, Y 93.4231, Z -8.0000, A 0.000, B 0.000, C 0.000 }
gfCNCPoint6[8882] = {X 457.0838, Y 93.0553, Z -8.0000, A 0.000, B 0.000, C 0.000 }
gfCNCPoint6[8883] = {X 457.9363, Y 92.8584, Z -8.0000, A 0.000, B 0.000, C 0.000 }
gfCNCPoint6[8884] = {X 457.9363, Y 85.5404, Z -8.0000, A 0.000, B 0.000, C 0.000 }
gfCNCPoint6[8885] = {X 444.8514, Y 80.4111, Z -8.0000, A 0.000, B 0.000, C 0.000 }
gfCNCPoint6[8886] = {X 419.9442, Y 96.5452, Z -8.0000, A 0.000, B 0.000, C 0.000 }
gfCNCPoint6[8887] = {X 419.9467, Y 97.0653, Z -8.0000, A 0.000, B 0.000, C 0.000 }
gfCNCPoint6[8888] = {X 419.9467, Y 98.0000, Z -8.0000, A 0.000, B 0.000, C 0.000 }
gfCNCPoint6[8889] = {X 419.8404, Y 98.9435, Z -8.0000, A 0.000, B 0.000, C 0.000 }
gfCNCPoint6[8890] = {X 419.5268, Y 99.8397, Z -8.0000, A 0.000, B 0.000, C 0.000 }
gfCNCPoint6[8891] = {X 419.0217, Y 100.6436, Z -8.0000, A 0.000, B 0.000, C 0.000 }
gfCNCPoint6[8892] = {X 418.3503, Y 101.3150, Z -8.0000, A 0.000, B 0.000, C 0.000 }
gfCNCPoint6[8893] = {X 417.5464, Y 101.8201, Z -8.0000, A 0.000, B 0.000, C 0.000 }
gfCNCPoint6[8894] = {X 416.6502, Y 102.1337, Z -8.0000, A 0.000, B 0.000, C 0.000 }
gfCNCPoint6[8895] = {X 415.7067, Y 102.2400, Z -8.0000, A 0.000, B 0.000, C 0.000 }
gfCNCPoint6[8896] = {X 396.4059, Y 102.2400, Z -8.0000, A 0.000, B 0.000, C 0.000 }
gfCNCPoint6[8897] = {X 395.4625, Y 102.1337, Z -8.0000, A 0.000, B 0.000, C 0.000 }
gfCNCPoint6[8898] = {X 394.5663, Y 101.8201, Z -8.0000, A 0.000, B 0.000, C 0.000 }
gfCNCPoint6[8899] = {X 393.7624, Y 101.3150, Z -8.0000, A 0.000, B 0.000, C 0.000 }
gfCNCPoint6[8900] = {X 393.0910, Y 100.6436, Z -8.0000, A 0.000, B 0.000, C 0.000 }
gfCNCPoint6[8901] = {X 392.5858, Y 99.8397, Z -8.0000, A 0.000, B 0.000, C 0.000 }
gfCNCPoint6[8902] = {X 392.2723, Y 98.9435, Z -8.0000, A 0.000, B 0.000, C 0.000 }
gfCNCPoint6[8903] = {X 392.1659, Y 98.0000, Z -8.0000, A 0.000, B 0.000, C 0.000 }
gfCNCPoint6[8904] = {X 392.1659, Y 97.0659, Z -8.0000, A 0.000, B 0.000, C 0.000 }
gfCNCPoint6[8905] = {X 392.2718, Y 96.1246, Z -8.0000, A 0.000, B 0.000, C 0.000 }
gfCNCPoint6[8906] = {X 392.5839, Y 95.2303, Z -8.0000, A 0.000, B 0.000, C 0.000 }
gfCNCPoint6[8907] = {X 393.0868, Y 94.4275, Z -8.0000, A 0.000, B 0.000, C 0.000 }
gfCNCPoint6[8908] = {X 393.7554, Y 93.7565, Z -8.0000, A 0.000, B 0.000, C 0.000 }
gfCNCPoint6[8909] = {X 394.5563, Y 93.2507, Z -8.0000, A 0.000, B 0.000, C 0.000 }
gfCNCPoint6[8910] = {X 395.4495, Y 92.9352, Z -8.0000, A 0.000, B 0.000, C 0.000 }
gfCNCPoint6[8911] = {X 396.3904, Y 92.8260, Z -8.0000, A 0.000, B 0.000, C 0.000 }
gfCNCPoint6[8912] = {X 397.3486, Y 92.7827, Z -8.0000, A 0.000, B 0.000, C 0.000 }
gfCNCPoint6[8913] = {X 398.3034, Y 92.6924, Z -8.0000, A 0.000, B 0.000, C 0.000 }
gfCNCPoint6[8914] = {X 398.9718, Y 92.5304, Z -8.0000, A 0.000, B 0.000, C 0.000 }
gfCNCPoint6[8915] = {X 399.5871, Y 92.2235, Z -8.0000, A 0.000, B 0.000, C 0.000 }
gfCNCPoint6[8916] = {X 413.8415, Y 83.0954, Z -8.0000, A 0.000, B 0.000, C 0.000 }
gfCNCPoint6[8917] = {X 411.6844, Y 79.7269, Z -8.0000, A 0.000, B 0.000, C 0.000 }
gfCNCPoint6[8918] = {X 413.8847, Y 83.1627, Z -8.0000, A 0.000, B 0.000, C 0.000 }
gfCNCPoint6[8919] = {X 428.4036, Y 73.8653, Z -8.0000, A 0.000, B 0.000, C 0.000 }
gfCNCPoint6[8920] = {X 403.8141, Y 64.2183, Z -8.0000, A 0.000, B 0.000, C 0.000 }
gfCNCPoint6[8921] = {X 402.1003, Y 63.6511, Z -8.0000, A 0.000, B 0.000, C 0.000 }
gfCNCPoint6[8922] = {X 400.3348, Y 63.2749, Z -8.0000, A 0.000, B 0.000, C 0.000 }
gfCNCPoint6[8923] = {X 398.5387, Y 63.0940, Z -8.0000, A 0.000, B 0.000, C 0.000 }
gfCNCPoint6[8924] = {X 397.6210, Y 62.9872, Z -8.0000, A 0.000, B 0.000, C 0.000 }
gfCNCPoint6[8925] = {X 396.7494, Y 62.6805, Z -8.0000, A 0.000, B 0.000, C 0.000 }
gfCNCPoint6[8926] = {X 395.9670, Y 62.1889, Z -8.0000, A 0.000, B 0.000, C 0.000 }
gfCNCPoint6[8927] = {X 395.3125, Y 61.5368, Z -8.0000, A 0.000, B 0.000, C 0.000 }
gfCNCPoint6[8928] = {X 394.8180, Y 60.7562, Z -8.0000, A 0.000, B 0.000, C 0.000 }
gfCNCPoint6[8929] = {X 394.5081, Y 59.8858, Z -8.0000, A 0.000, B 0.000, C 0.000 }
gfCNCPoint6[8930] = {X 394.3979, Y 58.9684, Z -8.0000, A 0.000, B 0.000, C 0.000 }
gfCNCPoint6[8931] = {X 394.3977, Y 58.0000, Z -8.0000, A 0.000, B 0.000, C 0.000 }
gfCNCPoint6[8932] = {X 394.5020, Y 57.0743, Z -8.0000, A 0.000, B 0.000, C 0.000 }
gfCNCPoint6[8933] = {X 394.8097, Y 56.1950, Z -8.0000, A 0.000, B 0.000, C 0.000 }
gfCNCPoint6[8934] = {X 395.3053, Y 55.4063, Z -8.0000, A 0.000, B 0.000, C 0.000 }
gfCNCPoint6[8935] = {X 395.9640, Y 54.7476, Z -8.0000, A 0.000, B 0.000, C 0.000 }
gfCNCPoint6[8936] = {X 396.7528, Y 54.2520, Z -8.0000, A 0.000, B 0.000, C 0.000 }
gfCNCPoint6[8937] = {X 397.6320, Y 53.9443, Z -8.0000, A 0.000, B 0.000, C 0.000 }
gfCNCPoint6[8938] = {X 398.5577, Y 53.8400, Z -8.0000, A 0.000, B 0.000, C 0.000 }
gfCNCPoint6[8939] = {X 419.4886, Y 53.8400, Z -8.0000, A 0.000, B 0.000, C 0.000 }
gfCNCPoint6[8940] = {X 420.4143, Y 53.9443, Z -8.0000, A 0.000, B 0.000, C 0.000 }
gfCNCPoint6[8941] = {X 421.2936, Y 54.2520, Z -8.0000, A 0.000, B 0.000, C 0.000 }
gfCNCPoint6[8942] = {X 422.0823, Y 54.7476, Z -8.0000, A 0.000, B 0.000, C 0.000 }
gfCNCPoint6[8943] = {X 422.7410, Y 55.4063, Z -8.0000, A 0.000, B 0.000, C 0.000 }
gfCNCPoint6[8944] = {X 423.2366, Y 56.1950, Z -8.0000, A 0.000, B 0.000, C 0.000 }
gfCNCPoint6[8945] = {X 423.5443, Y 57.0743, Z -8.0000, A 0.000, B 0.000, C 0.000 }
gfCNCPoint6[8946] = {X 423.6486, Y 58.0000, Z -8.0000, A 0.000, B 0.000, C 0.000 }
gfCNCPoint6[8947] = {X 423.6486, Y 58.3407, Z -8.0000, A 0.000, B 0.000, C 0.000 }
gfCNCPoint6[8948] = {X 429.5530, Y 60.6409, Z -8.0000, A 0.000, B 0.000, C 0.000 }
gfCNCPoint6[8949] = {X 458.0178, Y 71.9351, Z -8.0000, A 0.000, B 0.000, C 0.000 }
gfCNCPoint6[8950] = {X 458.0201, Y 63.0708, Z -8.0000, A 0.000, B 0.000, C 0.000 }
gfCNCPoint6[8951] = {X 457.9175, Y 63.0586, Z -8.0000, A 0.000, B 0.000, C 0.000 }
gfCNCPoint6[8952] = {X 457.8152, Y 63.0439, Z -8.0000, A 0.000, B 0.000, C 0.000 }
gfCNCPoint6[8953] = {X 456.8779, Y 62.7816, Z -8.0000, A 0.000, B 0.000, C 0.000 }
gfCNCPoint6[8954] = {X 456.0272, Y 62.3088, Z -8.0000, A 0.000, B 0.000, C 0.000 }
gfCNCPoint6[8955] = {X 455.3096, Y 61.6513, Z -8.0000, A 0.000, B 0.000, C 0.000 }
gfCNCPoint6[8956] = {X 454.7645, Y 60.8450, Z -8.0000, A 0.000, B 0.000, C 0.000 }
gfCNCPoint6[8957] = {X 454.4216, Y 59.9341, Z -8.0000, A 0.000, B 0.000, C 0.000 }
gfCNCPoint6[8958] = {X 454.2997, Y 58.9684, Z -8.0000, A 0.000, B 0.000, C 0.000 }
gfCNCPoint6[8959] = {X 454.2996, Y 58.0000, Z -8.0000, A 0.000, B 0.000, C 0.000 }
gfCNCPoint6[8960] = {X 454.4039, Y 57.0743, Z -8.0000, A 0.000, B 0.000, C 0.000 }
gfCNCPoint6[8961] = {X 454.7116, Y 56.1950, Z -8.0000, A 0.000, B 0.000, C 0.000 }
gfCNCPoint6[8962] = {X 455.2072, Y 55.4063, Z -8.0000, A 0.000, B 0.000, C 0.000 }
gfCNCPoint6[8963] = {X 455.8659, Y 54.7476, Z -8.0000, A 0.000, B 0.000, C 0.000 }
gfCNCPoint6[8964] = {X 456.6546, Y 54.2520, Z -8.0000, A 0.000, B 0.000, C 0.000 }
gfCNCPoint6[8965] = {X 457.5339, Y 53.9443, Z -8.0000, A 0.000, B 0.000, C 0.000 }
gfCNCPoint6[8966] = {X 458.4596, Y 53.8400, Z -8.0000, A 0.000, B 0.000, C 0.000 }
gfCNCPoint6[8967] = {X 475.0000, Y 53.8400, Z -8.0000, A 0.000, B 0.000, C 0.000 }
gfCNCPoint6[8968] = {X 475.9257, Y 53.9443, Z -8.0000, A 0.000, B 0.000, C 0.000 }
gfCNCPoint6[8969] = {X 476.8050, Y 54.2520, Z -8.0000, A 0.000, B 0.000, C 0.000 }
gfCNCPoint6[8970] = {X 477.5937, Y 54.7476, Z -8.0000, A 0.000, B 0.000, C 0.000 }
gfCNCPoint6[8971] = {X 478.2524, Y 55.4063, Z -8.0000, A 0.000, B 0.000, C 0.000 }
gfCNCPoint6[8972] = {X 478.7480, Y 56.1950, Z -8.0000, A 0.000, B 0.000, C 0.000 }
gfCNCPoint6[8973] = {X 479.0557, Y 57.0743, Z -8.0000, A 0.000, B 0.000, C 0.000 }
gfCNCPoint6[8974] = {X 479.1600, Y 58.0000, Z -8.0000, A 0.000, B 0.000, C 0.000 }
gfCNCPoint6[8975] = {X 479.1600, Y 58.9342, Z -8.0000, A 0.000, B 0.000, C 0.000 }
gfCNCPoint6[8976] = {X 479.0448, Y 59.9064, Z -8.0000, A 0.000, B 0.000, C 0.000 }
gfCNCPoint6[8977] = {X 478.7055, Y 60.8248, Z -8.0000, A 0.000, B 0.000, C 0.000 }
gfCNCPoint6[8978] = {X 478.1610, Y 61.6384, Z -8.0000, A 0.000, B 0.000, C 0.000 }
gfCNCPoint6[8979] = {X 477.4415, Y 62.3023, Z -8.0000, A 0.000, B 0.000, C 0.000 }
gfCNCPoint6[8980] = {X 476.5867, Y 62.7796, Z -8.0000, A 0.000, B 0.000, C 0.000 }
gfCNCPoint6[8981] = {X 475.6441, Y 63.0439, Z -8.0000, A 0.000, B 0.000, C 0.000 }
gfCNCPoint6[8982] = {X 475.5428, Y 63.0585, Z -8.0000, A 0.000, B 0.000, C 0.000 }
gfCNCPoint6[8983] = {X 475.4412, Y 63.0706, Z -8.0000, A 0.000, B 0.000, C 0.000 }
gfCNCPoint6[8984] = {X 475.4417, Y 92.8966, Z -8.0000, A 0.000, B 0.000, C 0.000 }
gfCNCPoint6[8985] = {X 475.8893, Y 93.0023, Z -8.0000, A 0.000, B 0.000, C 0.000 }
gfCNCPoint6[8986] = {X 476.3299, Y 93.1346, Z -8.0000, A 0.000, B 0.000, C 0.000 }
gfCNCPoint6[8987] = {X 477.1131, Y 93.4898, Z -8.0000, A 0.000, B 0.000, C 0.000 }
gfCNCPoint6[8988] = {X 477.8060, Y 93.9992, Z -8.0000, A 0.000, B 0.000, C 0.000 }
gfCNCPoint6[8989] = {X 478.3787, Y 94.6408, Z -8.0000, A 0.000, B 0.000, C 0.000 }
gfCNCPoint6[8990] = {X 478.8064, Y 95.3869, Z -8.0000, A 0.000, B 0.000, C 0.000 }
gfCNCPoint6[8991] = {X 479.0706, Y 96.2053, Z -8.0000, A 0.000, B 0.000, C 0.000 }
gfCNCPoint6[8992] = {X 479.1600, Y 97.0606, Z -8.0000, A 0.000, B 0.000, C 0.000 }
gfCNCPoint6[8993] = {X 479.1600, Y 98.0000, Z -8.0000, A 0.000, B 0.000, C 0.000 }
gfCNCPoint6[8994] = {X 479.0557, Y 98.9257, Z -8.0000, A 0.000, B 0.000, C 0.000 }
gfCNCPoint6[8995] = {X 478.7480, Y 99.8050, Z -8.0000, A 0.000, B 0.000, C 0.000 }
gfCNCPoint6[8996] = {X 478.2524, Y 100.5937, Z -8.0000, A 0.000, B 0.000, C 0.000 }
gfCNCPoint6[8997] = {X 477.5937, Y 101.2524, Z -8.0000, A 0.000, B 0.000, C 0.000 }
gfCNCPoint6[8998] = {X 476.8050, Y 101.7480, Z -8.0000, A 0.000, B 0.000, C 0.000 }
gfCNCPoint6[8999] = {X 475.9257, Y 102.0557, Z -8.0000, A 0.000, B 0.000, C 0.000 }
gfCNCPoint6[9000] = {X 475.0000, Y 102.1600, Z -8.0000, A 0.000, B 0.000, C 0.000 }
gfCNCPoint6[9001] = {X 458.4596, Y 102.1600, Z -8.0000, A 0.000, B 0.000, C 0.000 }
gfCNCPoint6[9002] = {X 457.5339, Y 102.0557, Z -8.0000, A 0.000, B 0.000, C 0.000 }
gfCNCPoint6[9003] = {X 456.6546, Y 101.7480, Z -8.0000, A 0.000, B 0.000, C 0.000 }
gfCNCPoint6[9004] = {X 455.8659, Y 101.2524, Z -8.0000, A 0.000, B 0.000, C 0.000 }
gfCNCPoint6[9005] = {X 455.2072, Y 100.5937, Z -8.0000, A 0.000, B 0.000, C 0.000 }
gfCNCPoint6[9006] = {X 454.7116, Y 99.8050, Z -8.0000, A 0.000, B 0.000, C 0.000 }
gfCNCPoint6[9007] = {X 454.4039, Y 98.9257, Z -8.0000, A 0.000, B 0.000, C 0.000 }
gfCNCPoint6[9008] = {X 454.2996, Y 98.0000, Z -8.0000, A 0.000, B 0.000, C 0.000 }
gfCNCPoint6[9009] = {X 454.2996, Y 97.0659, Z -8.0000, A 0.000, B 0.000, C 0.000 }
gfCNCPoint6[9010] = {X 454.3903, Y 96.2022, Z -8.0000, A 0.000, B 0.000, C 0.000 }
gfCNCPoint6[9011] = {X 454.6583, Y 95.3761, Z -8.0000, A 0.000, B 0.000, C 0.000 }
gfCNCPoint6[9012] = {X 455.0920, Y 94.6237, Z -8.0000, A 0.000, B 0.000, C 0.000 }
gfCNCPoint6[9013] = {X 455.6724, Y 93.9777, Z -8.0000, A 0.000, B 0.000, C 0.000 }
gfCNCPoint6[9014] = {X 456.3743, Y 93.4663, Z -8.0000, A 0.000, B 0.000, C 0.000 }
gfCNCPoint6[9015] = {X 457.1672, Y 93.1118, Z -8.0000, A 0.000, B 0.000, C 0.000 }
gfCNCPoint6[9016] = {X 458.0163, Y 92.9296, Z -8.0000, A 0.000, B 0.000, C 0.000 }
gfCNCPoint6[9017] = {X 458.0163, Y 85.4858, Z -8.0000, A 0.000, B 0.000, C 0.000 }
gfCNCPoint6[9018] = {X 444.8424, Y 80.3216, Z -8.0000, A 0.000, B 0.000, C 0.000 }
gfCNCPoint6[9019] = {X 419.8640, Y 96.5018, Z -8.0000, A 0.000, B 0.000, C 0.000 }
gfCNCPoint6[9020] = {X 419.8667, Y 97.0655, Z -8.0000, A 0.000, B 0.000, C 0.000 }
gfCNCPoint6[9021] = {X 419.8667, Y 98.0000, Z -8.0000, A 0.000, B 0.000, C 0.000 }
gfCNCPoint6[9022] = {X 419.7624, Y 98.9257, Z -8.0000, A 0.000, B 0.000, C 0.000 }
gfCNCPoint6[9023] = {X 419.4547, Y 99.8050, Z -8.0000, A 0.000, B 0.000, C 0.000 }
gfCNCPoint6[9024] = {X 418.9591, Y 100.5937, Z -8.0000, A 0.000, B 0.000, C 0.000 }
gfCNCPoint6[9025] = {X 418.3004, Y 101.2524, Z -8.0000, A 0.000, B 0.000, C 0.000 }
gfCNCPoint6[9026] = {X 417.5117, Y 101.7480, Z -8.0000, A 0.000, B 0.000, C 0.000 }
gfCNCPoint6[9027] = {X 416.6324, Y 102.0557, Z -8.0000, A 0.000, B 0.000, C 0.000 }
gfCNCPoint6[9028] = {X 415.7067, Y 102.1600, Z -8.0000, A 0.000, B 0.000, C 0.000 }
gfCNCPoint6[9029] = {X 396.4059, Y 102.1600, Z -8.0000, A 0.000, B 0.000, C 0.000 }
gfCNCPoint6[9030] = {X 395.4803, Y 102.0557, Z -8.0000, A 0.000, B 0.000, C 0.000 }
gfCNCPoint6[9031] = {X 394.6010, Y 101.7480, Z -8.0000, A 0.000, B 0.000, C 0.000 }
gfCNCPoint6[9032] = {X 393.8122, Y 101.2524, Z -8.0000, A 0.000, B 0.000, C 0.000 }
gfCNCPoint6[9033] = {X 393.1535, Y 100.5937, Z -8.0000, A 0.000, B 0.000, C 0.000 }
gfCNCPoint6[9034] = {X 392.6579, Y 99.8050, Z -8.0000, A 0.000, B 0.000, C 0.000 }
gfCNCPoint6[9035] = {X 392.3502, Y 98.9257, Z -8.0000, A 0.000, B 0.000, C 0.000 }
gfCNCPoint6[9036] = {X 392.2459, Y 98.0000, Z -8.0000, A 0.000, B 0.000, C 0.000 }
gfCNCPoint6[9037] = {X 392.2459, Y 97.0659, Z -8.0000, A 0.000, B 0.000, C 0.000 }
gfCNCPoint6[9038] = {X 392.3498, Y 96.1423, Z -8.0000, A 0.000, B 0.000, C 0.000 }
gfCNCPoint6[9039] = {X 392.6561, Y 95.2647, Z -8.0000, A 0.000, B 0.000, C 0.000 }
gfCNCPoint6[9040] = {X 393.1496, Y 94.4771, Z -8.0000, A 0.000, B 0.000, C 0.000 }
gfCNCPoint6[9041] = {X 393.8057, Y 93.8187, Z -8.0000, A 0.000, B 0.000, C 0.000 }
gfCNCPoint6[9042] = {X 394.5916, Y 93.3224, Z -8.0000, A 0.000, B 0.000, C 0.000 }
gfCNCPoint6[9043] = {X 395.4681, Y 93.0130, Z -8.0000, A 0.000, B 0.000, C 0.000 }
gfCNCPoint6[9044] = {X 396.3914, Y 92.9060, Z -8.0000, A 0.000, B 0.000, C 0.000 }
gfCNCPoint6[9045] = {X 397.3540, Y 92.8626, Z -8.0000, A 0.000, B 0.000, C 0.000 }
gfCNCPoint6[9046] = {X 398.3132, Y 92.7718, Z -8.0000, A 0.000, B 0.000, C 0.000 }
gfCNCPoint6[9047] = {X 398.9991, Y 92.6056, Z -8.0000, A 0.000, B 0.000, C 0.000 }
gfCNCPoint6[9048] = {X 399.6306, Y 92.2906, Z -8.0000, A 0.000, B 0.000, C 0.000 }
gfCNCPoint6[9049] = {X 413.8847, Y 83.1627, Z -8.0000, A 0.000, B 0.000, C 0.000 }
gfCNCPoint6[9050] = {X 411.7276, Y 79.7942, Z -8.0000, A 0.000, B 0.000, C 0.000 }
gfCNCPoint6[9051] = {X 413.9278, Y 83.2301, Z -8.0000, A 0.000, B 0.000, C 0.000 }
gfCNCPoint6[9052] = {X 428.5788, Y 73.8481, Z -8.0000, A 0.000, B 0.000, C 0.000 }
gfCNCPoint6[9053] = {X 403.8433, Y 64.1438, Z -8.0000, A 0.000, B 0.000, C 0.000 }
gfCNCPoint6[9054] = {X 402.1207, Y 63.5738, Z -8.0000, A 0.000, B 0.000, C 0.000 }
gfCNCPoint6[9055] = {X 400.3461, Y 63.1957, Z -8.0000, A 0.000, B 0.000, C 0.000 }
gfCNCPoint6[9056] = {X 398.5407, Y 63.0140, Z -8.0000, A 0.000, B 0.000, C 0.000 }
gfCNCPoint6[9057] = {X 397.6403, Y 62.9096, Z -8.0000, A 0.000, B 0.000, C 0.000 }
gfCNCPoint6[9058] = {X 396.7852, Y 62.6089, Z -8.0000, A 0.000, B 0.000, C 0.000 }
gfCNCPoint6[9059] = {X 396.0176, Y 62.1269, Z -8.0000, A 0.000, B 0.000, C 0.000 }
gfCNCPoint6[9060] = {X 395.3753, Y 61.4873, Z -8.0000, A 0.000, B 0.000, C 0.000 }
gfCNCPoint6[9061] = {X 394.8901, Y 60.7216, Z -8.0000, A 0.000, B 0.000, C 0.000 }
gfCNCPoint6[9062] = {X 394.5860, Y 59.8677, Z -8.0000, A 0.000, B 0.000, C 0.000 }
gfCNCPoint6[9063] = {X 394.4779, Y 58.9678, Z -8.0000, A 0.000, B 0.000, C 0.000 }
gfCNCPoint6[9064] = {X 394.4777, Y 58.0000, Z -8.0000, A 0.000, B 0.000, C 0.000 }
gfCNCPoint6[9065] = {X 394.5800, Y 57.0921, Z -8.0000, A 0.000, B 0.000, C 0.000 }
gfCNCPoint6[9066] = {X 394.8818, Y 56.2298, Z -8.0000, A 0.000, B 0.000, C 0.000 }
gfCNCPoint6[9067] = {X 395.3678, Y 55.4562, Z -8.0000, A 0.000, B 0.000, C 0.000 }
gfCNCPoint6[9068] = {X 396.0139, Y 54.8101, Z -8.0000, A 0.000, B 0.000, C 0.000 }
gfCNCPoint6[9069] = {X 396.7875, Y 54.3240, Z -8.0000, A 0.000, B 0.000, C 0.000 }
gfCNCPoint6[9070] = {X 397.6498, Y 54.0223, Z -8.0000, A 0.000, B 0.000, C 0.000 }
gfCNCPoint6[9071] = {X 398.5577, Y 53.9200, Z -8.0000, A 0.000, B 0.000, C 0.000 }
gfCNCPoint6[9072] = {X 419.4886, Y 53.9200, Z -8.0000, A 0.000, B 0.000, C 0.000 }
gfCNCPoint6[9073] = {X 420.3965, Y 54.0223, Z -8.0000, A 0.000, B 0.000, C 0.000 }
gfCNCPoint6[9074] = {X 421.2588, Y 54.3240, Z -8.0000, A 0.000, B 0.000, C 0.000 }
gfCNCPoint6[9075] = {X 422.0324, Y 54.8101, Z -8.0000, A 0.000, B 0.000, C 0.000 }
gfCNCPoint6[9076] = {X 422.6785, Y 55.4562, Z -8.0000, A 0.000, B 0.000, C 0.000 }
gfCNCPoint6[9077] = {X 423.1646, Y 56.2298, Z -8.0000, A 0.000, B 0.000, C 0.000 }
gfCNCPoint6[9078] = {X 423.4663, Y 57.0921, Z -8.0000, A 0.000, B 0.000, C 0.000 }
gfCNCPoint6[9079] = {X 423.5686, Y 58.0000, Z -8.0000, A 0.000, B 0.000, C 0.000 }
gfCNCPoint6[9080] = {X 423.5686, Y 58.3954, Z -8.0000, A 0.000, B 0.000, C 0.000 }
gfCNCPoint6[9081] = {X 429.5238, Y 60.7154, Z -8.0000, A 0.000, B 0.000, C 0.000 }
gfCNCPoint6[9082] = {X 458.0978, Y 72.0529, Z -8.0000, A 0.000, B 0.000, C 0.000 }
gfCNCPoint6[9083] = {X 458.1001, Y 62.9982, Z -8.0000, A 0.000, B 0.000, C 0.000 }
gfCNCPoint6[9084] = {X 457.9636, Y 62.9838, Z -8.0000, A 0.000, B 0.000, C 0.000 }
gfCNCPoint6[9085] = {X 457.8276, Y 62.9648, Z -8.0000, A 0.000, B 0.000, C 0.000 }
gfCNCPoint6[9086] = {X 456.9083, Y 62.7077, Z -8.0000, A 0.000, B 0.000, C 0.000 }
gfCNCPoint6[9087] = {X 456.0740, Y 62.2439, Z -8.0000, A 0.000, B 0.000, C 0.000 }
gfCNCPoint6[9088] = {X 455.3702, Y 61.5990, Z -8.0000, A 0.000, B 0.000, C 0.000 }
gfCNCPoint6[9089] = {X 454.8355, Y 60.8082, Z -8.0000, A 0.000, B 0.000, C 0.000 }
gfCNCPoint6[9090] = {X 454.4992, Y 59.9148, Z -8.0000, A 0.000, B 0.000, C 0.000 }
gfCNCPoint6[9091] = {X 454.3797, Y 58.9678, Z -8.0000, A 0.000, B 0.000, C 0.000 }
gfCNCPoint6[9092] = {X 454.3796, Y 58.0000, Z -8.0000, A 0.000, B 0.000, C 0.000 }
gfCNCPoint6[9093] = {X 454.4819, Y 57.0921, Z -8.0000, A 0.000, B 0.000, C 0.000 }
gfCNCPoint6[9094] = {X 454.7837, Y 56.2298, Z -8.0000, A 0.000, B 0.000, C 0.000 }
gfCNCPoint6[9095] = {X 455.2697, Y 55.4562, Z -8.0000, A 0.000, B 0.000, C 0.000 }
gfCNCPoint6[9096] = {X 455.9158, Y 54.8101, Z -8.0000, A 0.000, B 0.000, C 0.000 }
gfCNCPoint6[9097] = {X 456.6894, Y 54.3240, Z -8.0000, A 0.000, B 0.000, C 0.000 }
gfCNCPoint6[9098] = {X 457.5517, Y 54.0223, Z -8.0000, A 0.000, B 0.000, C 0.000 }
gfCNCPoint6[9099] = {X 458.4596, Y 53.9200, Z -8.0000, A 0.000, B 0.000, C 0.000 }
gfCNCPoint6[9100] = {X 475.0000, Y 53.9200, Z -8.0000, A 0.000, B 0.000, C 0.000 }
gfCNCPoint6[9101] = {X 475.9079, Y 54.0223, Z -8.0000, A 0.000, B 0.000, C 0.000 }
gfCNCPoint6[9102] = {X 476.7702, Y 54.3240, Z -8.0000, A 0.000, B 0.000, C 0.000 }
gfCNCPoint6[9103] = {X 477.5438, Y 54.8101, Z -8.0000, A 0.000, B 0.000, C 0.000 }
gfCNCPoint6[9104] = {X 478.1899, Y 55.4562, Z -8.0000, A 0.000, B 0.000, C 0.000 }
gfCNCPoint6[9105] = {X 478.6760, Y 56.2298, Z -8.0000, A 0.000, B 0.000, C 0.000 }
gfCNCPoint6[9106] = {X 478.9777, Y 57.0921, Z -8.0000, A 0.000, B 0.000, C 0.000 }
gfCNCPoint6[9107] = {X 479.0800, Y 58.0000, Z -8.0000, A 0.000, B 0.000, C 0.000 }
gfCNCPoint6[9108] = {X 479.0800, Y 58.9342, Z -8.0000, A 0.000, B 0.000, C 0.000 }
gfCNCPoint6[9109] = {X 478.9670, Y 59.8877, Z -8.0000, A 0.000, B 0.000, C 0.000 }
gfCNCPoint6[9110] = {X 478.6343, Y 60.7884, Z -8.0000, A 0.000, B 0.000, C 0.000 }
gfCNCPoint6[9111] = {X 478.1002, Y 61.5864, Z -8.0000, A 0.000, B 0.000, C 0.000 }
gfCNCPoint6[9112] = {X 477.3945, Y 62.2375, Z -8.0000, A 0.000, B 0.000, C 0.000 }
gfCNCPoint6[9113] = {X 476.5562, Y 62.7056, Z -8.0000, A 0.000, B 0.000, C 0.000 }
gfCNCPoint6[9114] = {X 475.6317, Y 62.9649, Z -8.0000, A 0.000, B 0.000, C 0.000 }
gfCNCPoint6[9115] = {X 475.4967, Y 62.9837, Z -8.0000, A 0.000, B 0.000, C 0.000 }
gfCNCPoint6[9116] = {X 475.3612, Y 62.9980, Z -8.0000, A 0.000, B 0.000, C 0.000 }
gfCNCPoint6[9117] = {X 475.3617, Y 92.9622, Z -8.0000, A 0.000, B 0.000, C 0.000 }
gfCNCPoint6[9118] = {X 475.8371, Y 93.0712, Z -8.0000, A 0.000, B 0.000, C 0.000 }
gfCNCPoint6[9119] = {X 476.3046, Y 93.2105, Z -8.0000, A 0.000, B 0.000, C 0.000 }
gfCNCPoint6[9120] = {X 477.0727, Y 93.5588, Z -8.0000, A 0.000, B 0.000, C 0.000 }
gfCNCPoint6[9121] = {X 477.7522, Y 94.0583, Z -8.0000, A 0.000, B 0.000, C 0.000 }
gfCNCPoint6[9122] = {X 478.3138, Y 94.6875, Z -8.0000, A 0.000, B 0.000, C 0.000 }
gfCNCPoint6[9123] = {X 478.7332, Y 95.4192, Z -8.0000, A 0.000, B 0.000, C 0.000 }
gfCNCPoint6[9124] = {X 478.9924, Y 96.2218, Z -8.0000, A 0.000, B 0.000, C 0.000 }
gfCNCPoint6[9125] = {X 479.0800, Y 97.0606, Z -8.0000, A 0.000, B 0.000, C 0.000 }
gfCNCPoint6[9126] = {X 479.0800, Y 98.0000, Z -8.0000, A 0.000, B 0.000, C 0.000 }
gfCNCPoint6[9127] = {X 478.9777, Y 98.9079, Z -8.0000, A 0.000, B 0.000, C 0.000 }
gfCNCPoint6[9128] = {X 478.6760, Y 99.7702, Z -8.0000, A 0.000, B 0.000, C 0.000 }
gfCNCPoint6[9129] = {X 478.1899, Y 100.5438, Z -8.0000, A 0.000, B 0.000, C 0.000 }
gfCNCPoint6[9130] = {X 477.5438, Y 101.1899, Z -8.0000, A 0.000, B 0.000, C 0.000 }
gfCNCPoint6[9131] = {X 476.7702, Y 101.6760, Z -8.0000, A 0.000, B 0.000, C 0.000 }
gfCNCPoint6[9132] = {X 475.9079, Y 101.9777, Z -8.0000, A 0.000, B 0.000, C 0.000 }
gfCNCPoint6[9133] = {X 475.0000, Y 102.0800, Z -8.0000, A 0.000, B 0.000, C 0.000 }
gfCNCPoint6[9134] = {X 458.4596, Y 102.0800, Z -8.0000, A 0.000, B 0.000, C 0.000 }
gfCNCPoint6[9135] = {X 457.5517, Y 101.9777, Z -8.0000, A 0.000, B 0.000, C 0.000 }
gfCNCPoint6[9136] = {X 456.6894, Y 101.6760, Z -8.0000, A 0.000, B 0.000, C 0.000 }
gfCNCPoint6[9137] = {X 455.9158, Y 101.1899, Z -8.0000, A 0.000, B 0.000, C 0.000 }
gfCNCPoint6[9138] = {X 455.2697, Y 100.5438, Z -8.0000, A 0.000, B 0.000, C 0.000 }
gfCNCPoint6[9139] = {X 454.7837, Y 99.7702, Z -8.0000, A 0.000, B 0.000, C 0.000 }
gfCNCPoint6[9140] = {X 454.4819, Y 98.9079, Z -8.0000, A 0.000, B 0.000, C 0.000 }
gfCNCPoint6[9141] = {X 454.3796, Y 98.0000, Z -8.0000, A 0.000, B 0.000, C 0.000 }
gfCNCPoint6[9142] = {X 454.3796, Y 97.0659, Z -8.0000, A 0.000, B 0.000, C 0.000 }
gfCNCPoint6[9143] = {X 454.4707, Y 96.2088, Z -8.0000, A 0.000, B 0.000, C 0.000 }
gfCNCPoint6[9144] = {X 454.7398, Y 95.3899, Z -8.0000, A 0.000, B 0.000, C 0.000 }
gfCNCPoint6[9145] = {X 455.1749, Y 94.6458, Z -8.0000, A 0.000, B 0.000, C 0.000 }
gfCNCPoint6[9146] = {X 455.7566, Y 94.0098, Z -8.0000, A 0.000, B 0.000, C 0.000 }
gfCNCPoint6[9147] = {X 456.4590, Y 93.5101, Z -8.0000, A 0.000, B 0.000, C 0.000 }
gfCNCPoint6[9148] = {X 457.2507, Y 93.1692, Z -8.0000, A 0.000, B 0.000, C 0.000 }
gfCNCPoint6[9149] = {X 458.0963, Y 93.0021, Z -8.0000, A 0.000, B 0.000, C 0.000 }
gfCNCPoint6[9150] = {X 458.0963, Y 85.4313, Z -8.0000, A 0.000, B 0.000, C 0.000 }
gfCNCPoint6[9151] = {X 444.8333, Y 80.2322, Z -8.0000, A 0.000, B 0.000, C 0.000 }
gfCNCPoint6[9152] = {X 419.7838, Y 96.4584, Z -8.0000, A 0.000, B 0.000, C 0.000 }
gfCNCPoint6[9153] = {X 419.7867, Y 97.0657, Z -8.0000, A 0.000, B 0.000, C 0.000 }
gfCNCPoint6[9154] = {X 419.7867, Y 98.0000, Z -8.0000, A 0.000, B 0.000, C 0.000 }
gfCNCPoint6[9155] = {X 419.6844, Y 98.9079, Z -8.0000, A 0.000, B 0.000, C 0.000 }
gfCNCPoint6[9156] = {X 419.3827, Y 99.7702, Z -8.0000, A 0.000, B 0.000, C 0.000 }
gfCNCPoint6[9157] = {X 418.8966, Y 100.5438, Z -8.0000, A 0.000, B 0.000, C 0.000 }
gfCNCPoint6[9158] = {X 418.2505, Y 101.1899, Z -8.0000, A 0.000, B 0.000, C 0.000 }
gfCNCPoint6[9159] = {X 417.4769, Y 101.6760, Z -8.0000, A 0.000, B 0.000, C 0.000 }
gfCNCPoint6[9160] = {X 416.6146, Y 101.9777, Z -8.0000, A 0.000, B 0.000, C 0.000 }
gfCNCPoint6[9161] = {X 415.7067, Y 102.0800, Z -8.0000, A 0.000, B 0.000, C 0.000 }
gfCNCPoint6[9162] = {X 396.4059, Y 102.0800, Z -8.0000, A 0.000, B 0.000, C 0.000 }
gfCNCPoint6[9163] = {X 395.4981, Y 101.9777, Z -8.0000, A 0.000, B 0.000, C 0.000 }
gfCNCPoint6[9164] = {X 394.6357, Y 101.6760, Z -8.0000, A 0.000, B 0.000, C 0.000 }
gfCNCPoint6[9165] = {X 393.8621, Y 101.1899, Z -8.0000, A 0.000, B 0.000, C 0.000 }
gfCNCPoint6[9166] = {X 393.2161, Y 100.5438, Z -8.0000, A 0.000, B 0.000, C 0.000 }
gfCNCPoint6[9167] = {X 392.7300, Y 99.7702, Z -8.0000, A 0.000, B 0.000, C 0.000 }
gfCNCPoint6[9168] = {X 392.4282, Y 98.9079, Z -8.0000, A 0.000, B 0.000, C 0.000 }
gfCNCPoint6[9169] = {X 392.3259, Y 98.0000, Z -8.0000, A 0.000, B 0.000, C 0.000 }
gfCNCPoint6[9170] = {X 392.3259, Y 97.0659, Z -8.0000, A 0.000, B 0.000, C 0.000 }
gfCNCPoint6[9171] = {X 392.4278, Y 96.1599, Z -8.0000, A 0.000, B 0.000, C 0.000 }
gfCNCPoint6[9172] = {X 392.7283, Y 95.2992, Z -8.0000, A 0.000, B 0.000, C 0.000 }
gfCNCPoint6[9173] = {X 393.2125, Y 94.5267, Z -8.0000, A 0.000, B 0.000, C 0.000 }
gfCNCPoint6[9174] = {X 393.8560, Y 93.8809, Z -8.0000, A 0.000, B 0.000, C 0.000 }
gfCNCPoint6[9175] = {X 394.6270, Y 93.3942, Z -8.0000, A 0.000, B 0.000, C 0.000 }
gfCNCPoint6[9176] = {X 395.4867, Y 93.0908, Z -8.0000, A 0.000, B 0.000, C 0.000 }
gfCNCPoint6[9177] = {X 396.3924, Y 92.9860, Z -8.0000, A 0.000, B 0.000, C 0.000 }
gfCNCPoint6[9178] = {X 397.3593, Y 92.9424, Z -8.0000, A 0.000, B 0.000, C 0.000 }
gfCNCPoint6[9179] = {X 398.3230, Y 92.8512, Z -8.0000, A 0.000, B 0.000, C 0.000 }
gfCNCPoint6[9180] = {X 399.0264, Y 92.6808, Z -8.0000, A 0.000, B 0.000, C 0.000 }
gfCNCPoint6[9181] = {X 399.6742, Y 92.3577, Z -8.0000, A 0.000, B 0.000, C 0.000 }
gfCNCPoint6[9182] = {X 413.9278, Y 83.2301, Z -8.0000, A 0.000, B 0.000, C 0.000 }
gfCNCPoint6[9183] = {X 411.7656, Y 79.8536, Z -8.0000, A 0.000, B 0.000, C 0.000 }
gfCNCPoint6[9184] = {X 411.7674, Y 79.8524, Z -8.0000, A 0.000, B 0.000, C 0.000 }
gfCNCPoint6[9185] = {X 413.9658, Y 83.2895, Z -8.0000, A 0.000, B 0.000, C 0.000 }
gfCNCPoint6[9186] = {X 428.7541, Y 73.8309, Z -8.0000, A 0.000, B 0.000, C 0.000 }
gfCNCPoint6[9187] = {X 403.8726, Y 64.0694, Z -8.0000, A 0.000, B 0.000, C 0.000 }
gfCNCPoint6[9188] = {X 402.1411, Y 63.4964, Z -8.0000, A 0.000, B 0.000, C 0.000 }
gfCNCPoint6[9189] = {X 400.3574, Y 63.1165, Z -8.0000, A 0.000, B 0.000, C 0.000 }
gfCNCPoint6[9190] = {X 398.5427, Y 62.9340, Z -8.0000, A 0.000, B 0.000, C 0.000 }
gfCNCPoint6[9191] = {X 397.6551, Y 62.8309, Z -8.0000, A 0.000, B 0.000, C 0.000 }
gfCNCPoint6[9192] = {X 396.8125, Y 62.5333, Z -8.0000, A 0.000, B 0.000, C 0.000 }
gfCNCPoint6[9193] = {X 396.0571, Y 62.0560, Z -8.0000, A 0.000, B 0.000, C 0.000 }
gfCNCPoint6[9194] = {X 395.4264, Y 61.4230, Z -8.0000, A 0.000, B 0.000, C 0.000 }
gfCNCPoint6[9195] = {X 394.9520, Y 60.6657, Z -8.0000, A 0.000, B 0.000, C 0.000 }
gfCNCPoint6[9196] = {X 394.6575, Y 59.8221, Z -8.0000, A 0.000, B 0.000, C 0.000 }
gfCNCPoint6[9197] = {X 394.5577, Y 58.9341, Z -8.0000, A 0.000, B 0.000, C 0.000 }
gfCNCPoint6[9198] = {X 394.5577, Y 58.0000, Z -8.0000, A 0.000, B 0.000, C 0.000 }
gfCNCPoint6[9199] = {X 394.6580, Y 57.1099, Z -8.0000, A 0.000, B 0.000, C 0.000 }
gfCNCPoint6[9200] = {X 394.9538, Y 56.2645, Z -8.0000, A 0.000, B 0.000, C 0.000 }
gfCNCPoint6[9201] = {X 395.4304, Y 55.5060, Z -8.0000, A 0.000, B 0.000, C 0.000 }
gfCNCPoint6[9202] = {X 396.0638, Y 54.8727, Z -8.0000, A 0.000, B 0.000, C 0.000 }
gfCNCPoint6[9203] = {X 396.8222, Y 54.3961, Z -8.0000, A 0.000, B 0.000, C 0.000 }
gfCNCPoint6[9204] = {X 397.6676, Y 54.1003, Z -8.0000, A 0.000, B 0.000, C 0.000 }
gfCNCPoint6[9205] = {X 398.5577, Y 54.0000, Z -8.0000, A 0.000, B 0.000, C 0.000 }
gfCNCPoint6[9206] = {X 419.4886, Y 54.0000, Z -8.0000, A 0.000, B 0.000, C 0.000 }
gfCNCPoint6[9207] = {X 420.3787, Y 54.1003, Z -8.0000, A 0.000, B 0.000, C 0.000 }
gfCNCPoint6[9208] = {X 421.2241, Y 54.3961, Z -8.0000, A 0.000, B 0.000, C 0.000 }
gfCNCPoint6[9209] = {X 421.9826, Y 54.8727, Z -8.0000, A 0.000, B 0.000, C 0.000 }
gfCNCPoint6[9210] = {X 422.6159, Y 55.5060, Z -8.0000, A 0.000, B 0.000, C 0.000 }
gfCNCPoint6[9211] = {X 423.0925, Y 56.2645, Z -8.0000, A 0.000, B 0.000, C 0.000 }
gfCNCPoint6[9212] = {X 423.3883, Y 57.1099, Z -8.0000, A 0.000, B 0.000, C 0.000 }
gfCNCPoint6[9213] = {X 423.4886, Y 58.0000, Z -8.0000, A 0.000, B 0.000, C 0.000 }
gfCNCPoint6[9214] = {X 423.4886, Y 58.4501, Z -8.0000, A 0.000, B 0.000, C 0.000 }
gfCNCPoint6[9215] = {X 429.4945, Y 60.7898, Z -8.0000, A 0.000, B 0.000, C 0.000 }
gfCNCPoint6[9216] = {X 458.1778, Y 72.1707, Z -8.0000, A 0.000, B 0.000, C 0.000 }
gfCNCPoint6[9217] = {X 458.1781, Y 63.0396, Z -8.0000, A 0.000, B 0.000, C 0.000 }
gfCNCPoint6[9218] = {X 458.1841, Y 62.9246, Z -8.0000, A 0.000, B 0.000, C 0.000 }
gfCNCPoint6[9219] = {X 458.0116, Y 62.9089, Z -8.0000, A 0.000, B 0.000, C 0.000 }
gfCNCPoint6[9220] = {X 457.8400, Y 62.8858, Z -8.0000, A 0.000, B 0.000, C 0.000 }
gfCNCPoint6[9221] = {X 456.9337, Y 62.6316, Z -8.0000, A 0.000, B 0.000, C 0.000 }
gfCNCPoint6[9222] = {X 456.1118, Y 62.1726, Z -8.0000, A 0.000, B 0.000, C 0.000 }
gfCNCPoint6[9223] = {X 455.4200, Y 61.5342, Z -8.0000, A 0.000, B 0.000, C 0.000 }
gfCNCPoint6[9224] = {X 454.8965, Y 60.7519, Z -8.0000, A 0.000, B 0.000, C 0.000 }
gfCNCPoint6[9225] = {X 454.5704, Y 59.8688, Z -8.0000, A 0.000, B 0.000, C 0.000 }
gfCNCPoint6[9226] = {X 454.4596, Y 58.9341, Z -8.0000, A 0.000, B 0.000, C 0.000 }
gfCNCPoint6[9227] = {X 454.4596, Y 58.0000, Z -8.0000, A 0.000, B 0.000, C 0.000 }
gfCNCPoint6[9228] = {X 454.5599, Y 57.1099, Z -8.0000, A 0.000, B 0.000, C 0.000 }
gfCNCPoint6[9229] = {X 454.8557, Y 56.2645, Z -8.0000, A 0.000, B 0.000, C 0.000 }
gfCNCPoint6[9230] = {X 455.3323, Y 55.5060, Z -8.0000, A 0.000, B 0.000, C 0.000 }
gfCNCPoint6[9231] = {X 455.9656, Y 54.8727, Z -8.0000, A 0.000, B 0.000, C 0.000 }
gfCNCPoint6[9232] = {X 456.7241, Y 54.3961, Z -8.0000, A 0.000, B 0.000, C 0.000 }
gfCNCPoint6[9233] = {X 457.5695, Y 54.1003, Z -8.0000, A 0.000, B 0.000, C 0.000 }
gfCNCPoint6[9234] = {X 458.4596, Y 54.0000, Z -8.0000, A 0.000, B 0.000, C 0.000 }
gfCNCPoint6[9235] = {X 475.0000, Y 54.0000, Z -8.0000, A 0.000, B 0.000, C 0.000 }
gfCNCPoint6[9236] = {X 475.8901, Y 54.1003, Z -8.0000, A 0.000, B 0.000, C 0.000 }
gfCNCPoint6[9237] = {X 476.7355, Y 54.3961, Z -8.0000, A 0.000, B 0.000, C 0.000 }
gfCNCPoint6[9238] = {X 477.4940, Y 54.8727, Z -8.0000, A 0.000, B 0.000, C 0.000 }
gfCNCPoint6[9239] = {X 478.1273, Y 55.5060, Z -8.0000, A 0.000, B 0.000, C 0.000 }
gfCNCPoint6[9240] = {X 478.6039, Y 56.2645, Z -8.0000, A 0.000, B 0.000, C 0.000 }
gfCNCPoint6[9241] = {X 478.8997, Y 57.1099, Z -8.0000, A 0.000, B 0.000, C 0.000 }
gfCNCPoint6[9242] = {X 479.0000, Y 58.0000, Z -8.0000, A 0.000, B 0.000, C 0.000 }
gfCNCPoint6[9243] = {X 478.9999, Y 58.9671, Z -8.0000, A 0.000, B 0.000, C 0.000 }
gfCNCPoint6[9244] = {X 478.8827, Y 59.8956, Z -8.0000, A 0.000, B 0.000, C 0.000 }
gfCNCPoint6[9245] = {X 478.5530, Y 60.7716, Z -8.0000, A 0.000, B 0.000, C 0.000 }
gfCNCPoint6[9246] = {X 478.0287, Y 61.5469, Z -8.0000, A 0.000, B 0.000, C 0.000 }
gfCNCPoint6[9247] = {X 477.3387, Y 62.1791, Z -8.0000, A 0.000, B 0.000, C 0.000 }
gfCNCPoint6[9248] = {X 476.5206, Y 62.6338, Z -8.0000, A 0.000, B 0.000, C 0.000 }
gfCNCPoint6[9249] = {X 475.6193, Y 62.8858, Z -8.0000, A 0.000, B 0.000, C 0.000 }
gfCNCPoint6[9250] = {X 475.4522, Y 62.9084, Z -8.0000, A 0.000, B 0.000, C 0.000 }
gfCNCPoint6[9251] = {X 475.2843, Y 62.9240, Z -8.0000, A 0.000, B 0.000, C 0.000 }
gfCNCPoint6[9252] = {X 475.2812, Y 63.2810, Z -8.0000, A 0.000, B 0.000, C 0.000 }
gfCNCPoint6[9253] = {X 475.2817, Y 93.0283, Z -8.0000, A 0.000, B 0.000, C 0.000 }
gfCNCPoint6[9254] = {X 475.7849, Y 93.1403, Z -8.0000, A 0.000, B 0.000, C 0.000 }
gfCNCPoint6[9255] = {X 476.2793, Y 93.2864, Z -8.0000, A 0.000, B 0.000, C 0.000 }
gfCNCPoint6[9256] = {X 477.0323, Y 93.6278, Z -8.0000, A 0.000, B 0.000, C 0.000 }
gfCNCPoint6[9257] = {X 477.6984, Y 94.1175, Z -8.0000, A 0.000, B 0.000, C 0.000 }
gfCNCPoint6[9258] = {X 478.2489, Y 94.7343, Z -8.0000, A 0.000, B 0.000, C 0.000 }
gfCNCPoint6[9259] = {X 478.6601, Y 95.4516, Z -8.0000, A 0.000, B 0.000, C 0.000 }
gfCNCPoint6[9260] = {X 478.9141, Y 96.2384, Z -8.0000, A 0.000, B 0.000, C 0.000 }
gfCNCPoint6[9261] = {X 479.0000, Y 97.0606, Z -8.0000, A 0.000, B 0.000, C 0.000 }
gfCNCPoint6[9262] = {X 479.0000, Y 98.0000, Z -8.0000, A 0.000, B 0.000, C 0.000 }
gfCNCPoint6[9263] = {X 478.8997, Y 98.8901, Z -8.0000, A 0.000, B 0.000, C 0.000 }
gfCNCPoint6[9264] = {X 478.6039, Y 99.7355, Z -8.0000, A 0.000, B 0.000, C 0.000 }
gfCNCPoint6[9265] = {X 478.1273, Y 100.4940, Z -8.0000, A 0.000, B 0.000, C 0.000 }
gfCNCPoint6[9266] = {X 477.4940, Y 101.1273, Z -8.0000, A 0.000, B 0.000, C 0.000 }
gfCNCPoint6[9267] = {X 476.7355, Y 101.6039, Z -8.0000, A 0.000, B 0.000, C 0.000 }
gfCNCPoint6[9268] = {X 475.8901, Y 101.8997, Z -8.0000, A 0.000, B 0.000, C 0.000 }
gfCNCPoint6[9269] = {X 475.0000, Y 102.0000, Z -8.0000, A 0.000, B 0.000, C 0.000 }
gfCNCPoint6[9270] = {X 458.4596, Y 102.0000, Z -8.0000, A 0.000, B 0.000, C 0.000 }
gfCNCPoint6[9271] = {X 457.5695, Y 101.8997, Z -8.0000, A 0.000, B 0.000, C 0.000 }
gfCNCPoint6[9272] = {X 456.7241, Y 101.6039, Z -8.0000, A 0.000, B 0.000, C 0.000 }
gfCNCPoint6[9273] = {X 455.9656, Y 101.1273, Z -8.0000, A 0.000, B 0.000, C 0.000 }
gfCNCPoint6[9274] = {X 455.3323, Y 100.4940, Z -8.0000, A 0.000, B 0.000, C 0.000 }
gfCNCPoint6[9275] = {X 454.8557, Y 99.7355, Z -8.0000, A 0.000, B 0.000, C 0.000 }
gfCNCPoint6[9276] = {X 454.5599, Y 98.8901, Z -8.0000, A 0.000, B 0.000, C 0.000 }
gfCNCPoint6[9277] = {X 454.4596, Y 98.0000, Z -8.0000, A 0.000, B 0.000, C 0.000 }
gfCNCPoint6[9278] = {X 454.4596, Y 97.0659, Z -8.0000, A 0.000, B 0.000, C 0.000 }
gfCNCPoint6[9279] = {X 454.5511, Y 96.2154, Z -8.0000, A 0.000, B 0.000, C 0.000 }
gfCNCPoint6[9280] = {X 454.8213, Y 95.4037, Z -8.0000, A 0.000, B 0.000, C 0.000 }
gfCNCPoint6[9281] = {X 455.2580, Y 94.6681, Z -8.0000, A 0.000, B 0.000, C 0.000 }
gfCNCPoint6[9282] = {X 455.8411, Y 94.0422, Z -8.0000, A 0.000, B 0.000, C 0.000 }
gfCNCPoint6[9283] = {X 456.5439, Y 93.5545, Z -8.0000, A 0.000, B 0.000, C 0.000 }
gfCNCPoint6[9284] = {X 457.3344, Y 93.2275, Z -8.0000, A 0.000, B 0.000, C 0.000 }
gfCNCPoint6[9285] = {X 458.1763, Y 93.0760, Z -8.0000, A 0.000, B 0.000, C 0.000 }
gfCNCPoint6[9286] = {X 458.1763, Y 85.3767, Z -8.0000, A 0.000, B 0.000, C 0.000 }
gfCNCPoint6[9287] = {X 444.8243, Y 80.1427, Z -8.0000, A 0.000, B 0.000, C 0.000 }
gfCNCPoint6[9288] = {X 419.7036, Y 96.4151, Z -8.0000, A 0.000, B 0.000, C 0.000 }
gfCNCPoint6[9289] = {X 419.7067, Y 97.0659, Z -8.0000, A 0.000, B 0.000, C 0.000 }
gfCNCPoint6[9290] = {X 419.7067, Y 98.0000, Z -8.0000, A 0.000, B 0.000, C 0.000 }
gfCNCPoint6[9291] = {X 419.6064, Y 98.8901, Z -8.0000, A 0.000, B 0.000, C 0.000 }
gfCNCPoint6[9292] = {X 419.3106, Y 99.7355, Z -8.0000, A 0.000, B 0.000, C 0.000 }
gfCNCPoint6[9293] = {X 418.8340, Y 100.4940, Z -8.0000, A 0.000, B 0.000, C 0.000 }
gfCNCPoint6[9294] = {X 418.2007, Y 101.1273, Z -8.0000, A 0.000, B 0.000, C 0.000 }
gfCNCPoint6[9295] = {X 417.4422, Y 101.6039, Z -8.0000, A 0.000, B 0.000, C 0.000 }
gfCNCPoint6[9296] = {X 416.5968, Y 101.8997, Z -8.0000, A 0.000, B 0.000, C 0.000 }
gfCNCPoint6[9297] = {X 415.7067, Y 102.0000, Z -8.0000, A 0.000, B 0.000, C 0.000 }
gfCNCPoint6[9298] = {X 396.4059, Y 102.0000, Z -8.0000, A 0.000, B 0.000, C 0.000 }
gfCNCPoint6[9299] = {X 395.5159, Y 101.8997, Z -8.0000, A 0.000, B 0.000, C 0.000 }
gfCNCPoint6[9300] = {X 394.6704, Y 101.6039, Z -8.0000, A 0.000, B 0.000, C 0.000 }
gfCNCPoint6[9301] = {X 393.9120, Y 101.1273, Z -8.0000, A 0.000, B 0.000, C 0.000 }
gfCNCPoint6[9302] = {X 393.2786, Y 100.4940, Z -8.0000, A 0.000, B 0.000, C 0.000 }
gfCNCPoint6[9303] = {X 392.8021, Y 99.7355, Z -8.0000, A 0.000, B 0.000, C 0.000 }
gfCNCPoint6[9304] = {X 392.5062, Y 98.8901, Z -8.0000, A 0.000, B 0.000, C 0.000 }
gfCNCPoint6[9305] = {X 392.4059, Y 98.0000, Z -8.0000, A 0.000, B 0.000, C 0.000 }
gfCNCPoint6[9306] = {X 392.4059, Y 97.0659, Z -8.0000, A 0.000, B 0.000, C 0.000 }
gfCNCPoint6[9307] = {X 392.5058, Y 96.1776, Z -8.0000, A 0.000, B 0.000, C 0.000 }
gfCNCPoint6[9308] = {X 392.8005, Y 95.3337, Z -8.0000, A 0.000, B 0.000, C 0.000 }
gfCNCPoint6[9309] = {X 393.2753, Y 94.5762, Z -8.0000, A 0.000, B 0.000, C 0.000 }
gfCNCPoint6[9310] = {X 393.9064, Y 93.9431, Z -8.0000, A 0.000, B 0.000, C 0.000 }
gfCNCPoint6[9311] = {X 394.6623, Y 93.4660, Z -8.0000, A 0.000, B 0.000, C 0.000 }
gfCNCPoint6[9312] = {X 395.5053, Y 93.1686, Z -8.0000, A 0.000, B 0.000, C 0.000 }
gfCNCPoint6[9313] = {X 396.3933, Y 93.0660, Z -8.0000, A 0.000, B 0.000, C 0.000 }
gfCNCPoint6[9314] = {X 397.3647, Y 93.0222, Z -8.0000, A 0.000, B 0.000, C 0.000 }
gfCNCPoint6[9315] = {X 398.3327, Y 92.9306, Z -8.0000, A 0.000, B 0.000, C 0.000 }
gfCNCPoint6[9316] = {X 399.0538, Y 92.7560, Z -8.0000, A 0.000, B 0.000, C 0.000 }
gfCNCPoint6[9317] = {X 399.7177, Y 92.4248, Z -8.0000, A 0.000, B 0.000, C 0.000 }
gfCNCPoint6[9318] = {X 404.3150, Y 89.4621, Z -8.0000, A 0.000, B 0.000, C 0.000 }
gfCNCPoint6[9319] = {X 413.9658, Y 83.2895, Z -8.0000, A 0.000, B 0.000, C 0.000 }
gfCNCPoint6[9320] = {X 411.7674, Y 79.8524, Z -8.0000, A 0.000, B 0.000, C 0.000 }
gfCNCPoint6[9321] = {X 411.7674, Y 79.8524, Z -5.0000, A 0.000, B 0.000, C 0.000 }
gfCNCPoint6[9322] = {X 411.7674, Y 79.8524, Z 11.0000, A 0.000, B 0.000, C 0.000 }
gfCNCPoint6[9323] = {X 466.3120, Y 28.5934, Z 11.0000, A 0.000, B 0.000, C 0.000 }
gfCNCPoint6[9324] = {X 466.3120, Y 28.5934, Z -5.0000, A 0.000, B 0.000, C 0.000 }
gfCNCPoint6[9325] = {X 466.3120, Y 28.5934, Z -8.0000, A 0.000, B 0.000, C 0.000 }
gfCNCPoint6[9326] = {X 462.2320, Y 28.5935, Z -8.0000, A 0.000, B 0.000, C 0.000 }
gfCNCPoint6[9327] = {X 462.2323, Y 40.9144, Z -8.0000, A 0.000, B 0.000, C 0.000 }
gfCNCPoint6[9328] = {X 462.2406, Y 40.9213, Z -8.0000, A 0.000, B 0.000, C 0.000 }
gfCNCPoint6[9329] = {X 462.8750, Y 41.5917, Z -8.0000, A 0.000, B 0.000, C 0.000 }
gfCNCPoint6[9330] = {X 463.3525, Y 42.3816, Z -8.0000, A 0.000, B 0.000, C 0.000 }
gfCNCPoint6[9331] = {X 463.6513, Y 43.2549, Z -8.0000, A 0.000, B 0.000, C 0.000 }
gfCNCPoint6[9332] = {X 463.7578, Y 44.1718, Z -8.0000, A 0.000, B 0.000, C 0.000 }
gfCNCPoint6[9333] = {X 463.7579, Y 45.0000, Z -8.0000, A 0.000, B 0.000, C 0.000 }
gfCNCPoint6[9334] = {X 463.6496, Y 45.9613, Z -8.0000, A 0.000, B 0.000, C 0.000 }
gfCNCPoint6[9335] = {X 463.3301, Y 46.8744, Z -8.0000, A 0.000, B 0.000, C 0.000 }
gfCNCPoint6[9336] = {X 462.8155, Y 47.6935, Z -8.0000, A 0.000, B 0.000, C 0.000 }
gfCNCPoint6[9337] = {X 462.1314, Y 48.3775, Z -8.0000, A 0.000, B 0.000, C 0.000 }
gfCNCPoint6[9338] = {X 461.3123, Y 48.8922, Z -8.0000, A 0.000, B 0.000, C 0.000 }
gfCNCPoint6[9339] = {X 460.3992, Y 49.2117, Z -8.0000, A 0.000, B 0.000, C 0.000 }
gfCNCPoint6[9340] = {X 459.4379, Y 49.3200, Z -8.0000, A 0.000, B 0.000, C 0.000 }
gfCNCPoint6[9341] = {X 452.9945, Y 49.3200, Z -8.0000, A 0.000, B 0.000, C 0.000 }
gfCNCPoint6[9342] = {X 452.0380, Y 49.2128, Z -8.0000, A 0.000, B 0.000, C 0.000 }
gfCNCPoint6[9343] = {X 451.1291, Y 48.8965, Z -8.0000, A 0.000, B 0.000, C 0.000 }
gfCNCPoint6[9344] = {X 450.3127, Y 48.3868, Z -8.0000, A 0.000, B 0.000, C 0.000 }
gfCNCPoint6[9345] = {X 449.6294, Y 47.7091, Z -8.0000, A 0.000, B 0.000, C 0.000 }
gfCNCPoint6[9346] = {X 449.1132, Y 46.8968, Z -8.0000, A 0.000, B 0.000, C 0.000 }
gfCNCPoint6[9347] = {X 448.7895, Y 45.9905, Z -8.0000, A 0.000, B 0.000, C 0.000 }
gfCNCPoint6[9348] = {X 448.6746, Y 45.0349, Z -8.0000, A 0.000, B 0.000, C 0.000 }
gfCNCPoint6[9349] = {X 448.6749, Y 44.1494, Z -8.0000, A 0.000, B 0.000, C 0.000 }
gfCNCPoint6[9350] = {X 448.7853, Y 43.2364, Z -8.0000, A 0.000, B 0.000, C 0.000 }
gfCNCPoint6[9351] = {X 449.0865, Y 42.3675, Z -8.0000, A 0.000, B 0.000, C 0.000 }
gfCNCPoint6[9352] = {X 449.5648, Y 41.5821, Z -8.0000, A 0.000, B 0.000, C 0.000 }
gfCNCPoint6[9353] = {X 450.1984, Y 40.9157, Z -8.0000, A 0.000, B 0.000, C 0.000 }
gfCNCPoint6[9354] = {X 450.1984, Y 34.4738, Z -8.0000, A 0.000, B 0.000, C 0.000 }
gfCNCPoint6[9355] = {X 447.4757, Y 34.4738, Z -8.0000, A 0.000, B 0.000, C 0.000 }
gfCNCPoint6[9356] = {X 443.1903, Y 42.8182, Z -8.0000, A 0.000, B 0.000, C 0.000 }
gfCNCPoint6[9357] = {X 443.1950, Y 42.8315, Z -8.0000, A 0.000, B 0.000, C 0.000 }
gfCNCPoint6[9358] = {X 443.3606, Y 43.4920, Z -8.0000, A 0.000, B 0.000, C 0.000 }
gfCNCPoint6[9359] = {X 443.4203, Y 44.1703, Z -8.0000, A 0.000, B 0.000, C 0.000 }
gfCNCPoint6[9360] = {X 443.4205, Y 45.0000, Z -8.0000, A 0.000, B 0.000, C 0.000 }
gfCNCPoint6[9361] = {X 443.3122, Y 45.9613, Z -8.0000, A 0.000, B 0.000, C 0.000 }
gfCNCPoint6[9362] = {X 442.9927, Y 46.8744, Z -8.0000, A 0.000, B 0.000, C 0.000 }
gfCNCPoint6[9363] = {X 442.4780, Y 47.6935, Z -8.0000, A 0.000, B 0.000, C 0.000 }
gfCNCPoint6[9364] = {X 441.7939, Y 48.3775, Z -8.0000, A 0.000, B 0.000, C 0.000 }
gfCNCPoint6[9365] = {X 440.9748, Y 48.8922, Z -8.0000, A 0.000, B 0.000, C 0.000 }
gfCNCPoint6[9366] = {X 440.0618, Y 49.2117, Z -8.0000, A 0.000, B 0.000, C 0.000 }
gfCNCPoint6[9367] = {X 439.1005, Y 49.3200, Z -8.0000, A 0.000, B 0.000, C 0.000 }
gfCNCPoint6[9368] = {X 432.5144, Y 49.3200, Z -8.0000, A 0.000, B 0.000, C 0.000 }
gfCNCPoint6[9369] = {X 431.5531, Y 49.2117, Z -8.0000, A 0.000, B 0.000, C 0.000 }
gfCNCPoint6[9370] = {X 430.6401, Y 48.8922, Z -8.0000, A 0.000, B 0.000, C 0.000 }
gfCNCPoint6[9371] = {X 429.8210, Y 48.3775, Z -8.0000, A 0.000, B 0.000, C 0.000 }
gfCNCPoint6[9372] = {X 429.1369, Y 47.6935, Z -8.0000, A 0.000, B 0.000, C 0.000 }
gfCNCPoint6[9373] = {X 428.6223, Y 46.8744, Z -8.0000, A 0.000, B 0.000, C 0.000 }
gfCNCPoint6[9374] = {X 428.3027, Y 45.9614, Z -8.0000, A 0.000, B 0.000, C 0.000 }
gfCNCPoint6[9375] = {X 428.1944, Y 45.0001, Z -8.0000, A 0.000, B 0.000, C 0.000 }
gfCNCPoint6[9376] = {X 428.1948, Y 44.1494, Z -8.0000, A 0.000, B 0.000, C 0.000 }
gfCNCPoint6[9377] = {X 428.2925, Y 43.2935, Z -8.0000, A 0.000, B 0.000, C 0.000 }
gfCNCPoint6[9378] = {X 428.5580, Y 42.4740, Z -8.0000, A 0.000, B 0.000, C 0.000 }
gfCNCPoint6[9379] = {X 428.9809, Y 41.7236, Z -8.0000, A 0.000, B 0.000, C 0.000 }
gfCNCPoint6[9380] = {X 429.5442, Y 41.0719, Z -8.0000, A 0.000, B 0.000, C 0.000 }
gfCNCPoint6[9381] = {X 430.2256, Y 40.5449, Z -8.0000, A 0.000, B 0.000, C 0.000 }
gfCNCPoint6[9382] = {X 430.9981, Y 40.1637, Z -8.0000, A 0.000, B 0.000, C 0.000 }
gfCNCPoint6[9383] = {X 434.9867, Y 32.3564, Z -8.0000, A 0.000, B 0.000, C 0.000 }
gfCNCPoint6[9384] = {X 433.8230, Y 31.5744, Z -8.0000, A 0.000, B 0.000, C 0.000 }
gfCNCPoint6[9385] = {X 432.7647, Y 30.6548, Z -8.0000, A 0.000, B 0.000, C 0.000 }
gfCNCPoint6[9386] = {X 431.8281, Y 29.6115, Z -8.0000, A 0.000, B 0.000, C 0.000 }
gfCNCPoint6[9387] = {X 431.0276, Y 28.4605, Z -8.0000, A 0.000, B 0.000, C 0.000 }
gfCNCPoint6[9388] = {X 430.3752, Y 27.2195, Z -8.0000, A 0.000, B 0.000, C 0.000 }
gfCNCPoint6[9389] = {X 429.8811, Y 25.9074, Z -8.0000, A 0.000, B 0.000, C 0.000 }
gfCNCPoint6[9390] = {X 429.4495, Y 24.0610, Z -8.0000, A 0.000, B 0.000, C 0.000 }
gfCNCPoint6[9391] = {X 429.2322, Y 22.1772, Z -8.0000, A 0.000, B 0.000, C 0.000 }
gfCNCPoint6[9392] = {X 429.2319, Y 20.2809, Z -8.0000, A 0.000, B 0.000, C 0.000 }
gfCNCPoint6[9393] = {X 429.4489, Y 18.3971, Z -8.0000, A 0.000, B 0.000, C 0.000 }
gfCNCPoint6[9394] = {X 429.8801, Y 16.5505, Z -8.0000, A 0.000, B 0.000, C 0.000 }
gfCNCPoint6[9395] = {X 430.4498, Y 15.0194, Z -8.0000, A 0.000, B 0.000, C 0.000 }
gfCNCPoint6[9396] = {X 431.2251, Y 13.5813, Z -8.0000, A 0.000, B 0.000, C 0.000 }
gfCNCPoint6[9397] = {X 432.1912, Y 12.2638, Z -8.0000, A 0.000, B 0.000, C 0.000 }
gfCNCPoint6[9398] = {X 433.3295, Y 11.0919, Z -8.0000, A 0.000, B 0.000, C 0.000 }
gfCNCPoint6[9399] = {X 434.6185, Y 10.0880, Z -8.0000, A 0.000, B 0.000, C 0.000 }
gfCNCPoint6[9400] = {X 436.0334, Y 9.2713, Z -8.0000, A 0.000, B 0.000, C 0.000 }
gfCNCPoint6[9401] = {X 437.5474, Y 8.6573, Z -8.0000, A 0.000, B 0.000, C 0.000 }
gfCNCPoint6[9402] = {X 439.1316, Y 8.2578, Z -8.0000, A 0.000, B 0.000, C 0.000 }
gfCNCPoint6[9403] = {X 441.2286, Y 7.9675, Z -8.0000, A 0.000, B 0.000, C 0.000 }
gfCNCPoint6[9404] = {X 443.3436, Y 7.8733, Z -8.0000, A 0.000, B 0.000, C 0.000 }
gfCNCPoint6[9405] = {X 444.0357, Y 7.8692, Z -8.0000, A 0.000, B 0.000, C 0.000 }
gfCNCPoint6[9406] = {X 459.4469, Y 7.8692, Z -8.0000, A 0.000, B 0.000, C 0.000 }
gfCNCPoint6[9407] = {X 460.4062, Y 7.9773, Z -8.0000, A 0.000, B 0.000, C 0.000 }
gfCNCPoint6[9408] = {X 461.3174, Y 8.2962, Z -8.0000, A 0.000, B 0.000, C 0.000 }
gfCNCPoint6[9409] = {X 462.1348, Y 8.8098, Z -8.0000, A 0.000, B 0.000, C 0.000 }
gfCNCPoint6[9410] = {X 462.8174, Y 9.4924, Z -8.0000, A 0.000, B 0.000, C 0.000 }
gfCNCPoint6[9411] = {X 463.3310, Y 10.3098, Z -8.0000, A 0.000, B 0.000, C 0.000 }
gfCNCPoint6[9412] = {X 463.6499, Y 11.2210, Z -8.0000, A 0.000, B 0.000, C 0.000 }
gfCNCPoint6[9413] = {X 463.7579, Y 12.1803, Z -8.0000, A 0.000, B 0.000, C 0.000 }
gfCNCPoint6[9414] = {X 463.7579, Y 12.9782, Z -8.0000, A 0.000, B 0.000, C 0.000 }
gfCNCPoint6[9415] = {X 463.6567, Y 13.9076, Z -8.0000, A 0.000, B 0.000, C 0.000 }
gfCNCPoint6[9416] = {X 463.3578, Y 14.7935, Z -8.0000, A 0.000, B 0.000, C 0.000 }
gfCNCPoint6[9417] = {X 462.8753, Y 15.5943, Z -8.0000, A 0.000, B 0.000, C 0.000 }
gfCNCPoint6[9418] = {X 462.2318, Y 16.2725, Z -8.0000, A 0.000, B 0.000, C 0.000 }
gfCNCPoint6[9419] = {X 462.2320, Y 28.5935, Z -8.0000, A 0.000, B 0.000, C 0.000 }
gfCNCPoint6[9420] = {X 466.2320, Y 28.5934, Z -8.0000, A 0.000, B 0.000, C 0.000 }
gfCNCPoint6[9421] = {X 462.1520, Y 28.5935, Z -8.0000, A 0.000, B 0.000, C 0.000 }
gfCNCPoint6[9422] = {X 462.1523, Y 40.9520, Z -8.0000, A 0.000, B 0.000, C 0.000 }
gfCNCPoint6[9423] = {X 462.1891, Y 40.9825, Z -8.0000, A 0.000, B 0.000, C 0.000 }
gfCNCPoint6[9424] = {X 462.8116, Y 41.6405, Z -8.0000, A 0.000, B 0.000, C 0.000 }
gfCNCPoint6[9425] = {X 463.2801, Y 42.4157, Z -8.0000, A 0.000, B 0.000, C 0.000 }
gfCNCPoint6[9426] = {X 463.5733, Y 43.2727, Z -8.0000, A 0.000, B 0.000, C 0.000 }
gfCNCPoint6[9427] = {X 463.6778, Y 44.1724, Z -8.0000, A 0.000, B 0.000, C 0.000 }
gfCNCPoint6[9428] = {X 463.6779, Y 45.0000, Z -8.0000, A 0.000, B 0.000, C 0.000 }
gfCNCPoint6[9429] = {X 463.5716, Y 45.9435, Z -8.0000, A 0.000, B 0.000, C 0.000 }
gfCNCPoint6[9430] = {X 463.2580, Y 46.8397, Z -8.0000, A 0.000, B 0.000, C 0.000 }
gfCNCPoint6[9431] = {X 462.7529, Y 47.6436, Z -8.0000, A 0.000, B 0.000, C 0.000 }
gfCNCPoint6[9432] = {X 462.0815, Y 48.3150, Z -8.0000, A 0.000, B 0.000, C 0.000 }
gfCNCPoint6[9433] = {X 461.2776, Y 48.8201, Z -8.0000, A 0.000, B 0.000, C 0.000 }
gfCNCPoint6[9434] = {X 460.3814, Y 49.1337, Z -8.0000, A 0.000, B 0.000, C 0.000 }
gfCNCPoint6[9435] = {X 459.4379, Y 49.2400, Z -8.0000, A 0.000, B 0.000, C 0.000 }
gfCNCPoint6[9436] = {X 452.9945, Y 49.2400, Z -8.0000, A 0.000, B 0.000, C 0.000 }
gfCNCPoint6[9437] = {X 452.0558, Y 49.1348, Z -8.0000, A 0.000, B 0.000, C 0.000 }
gfCNCPoint6[9438] = {X 451.1636, Y 48.8243, Z -8.0000, A 0.000, B 0.000, C 0.000 }
gfCNCPoint6[9439] = {X 450.3624, Y 48.3241, Z -8.0000, A 0.000, B 0.000, C 0.000 }
gfCNCPoint6[9440] = {X 449.6918, Y 47.6589, Z -8.0000, A 0.000, B 0.000, C 0.000 }
gfCNCPoint6[9441] = {X 449.1851, Y 46.8617, Z -8.0000, A 0.000, B 0.000, C 0.000 }
gfCNCPoint6[9442] = {X 448.8674, Y 45.9721, Z -8.0000, A 0.000, B 0.000, C 0.000 }
gfCNCPoint6[9443] = {X 448.7546, Y 45.0343, Z -8.0000, A 0.000, B 0.000, C 0.000 }
gfCNCPoint6[9444] = {X 448.7549, Y 44.1505, Z -8.0000, A 0.000, B 0.000, C 0.000 }
gfCNCPoint6[9445] = {X 448.8654, Y 43.2454, Z -8.0000, A 0.000, B 0.000, C 0.000 }
gfCNCPoint6[9446] = {X 449.1668, Y 42.3850, Z -8.0000, A 0.000, B 0.000, C 0.000 }
gfCNCPoint6[9447] = {X 449.6452, Y 41.6088, Z -8.0000, A 0.000, B 0.000, C 0.000 }
gfCNCPoint6[9448] = {X 450.2784, Y 40.9529, Z -8.0000, A 0.000, B 0.000, C 0.000 }
gfCNCPoint6[9449] = {X 450.2784, Y 34.3938, Z -8.0000, A 0.000, B 0.000, C 0.000 }
gfCNCPoint6[9450] = {X 447.4268, Y 34.3938, Z -8.0000, A 0.000, B 0.000, C 0.000 }
gfCNCPoint6[9451] = {X 443.1033, Y 42.8124, Z -8.0000, A 0.000, B 0.000, C 0.000 }
gfCNCPoint6[9452] = {X 443.1194, Y 42.8577, Z -8.0000, A 0.000, B 0.000, C 0.000 }
gfCNCPoint6[9453] = {X 443.2818, Y 43.5056, Z -8.0000, A 0.000, B 0.000, C 0.000 }
gfCNCPoint6[9454] = {X 443.3403, Y 44.1710, Z -8.0000, A 0.000, B 0.000, C 0.000 }
gfCNCPoint6[9455] = {X 443.3405, Y 45.0000, Z -8.0000, A 0.000, B 0.000, C 0.000 }
gfCNCPoint6[9456] = {X 443.2342, Y 45.9435, Z -8.0000, A 0.000, B 0.000, C 0.000 }
gfCNCPoint6[9457] = {X 442.9206, Y 46.8397, Z -8.0000, A 0.000, B 0.000, C 0.000 }
gfCNCPoint6[9458] = {X 442.4154, Y 47.6436, Z -8.0000, A 0.000, B 0.000, C 0.000 }
gfCNCPoint6[9459] = {X 441.7441, Y 48.3150, Z -8.0000, A 0.000, B 0.000, C 0.000 }
gfCNCPoint6[9460] = {X 440.9401, Y 48.8201, Z -8.0000, A 0.000, B 0.000, C 0.000 }
gfCNCPoint6[9461] = {X 440.0440, Y 49.1337, Z -8.0000, A 0.000, B 0.000, C 0.000 }
gfCNCPoint6[9462] = {X 439.1005, Y 49.2400, Z -8.0000, A 0.000, B 0.000, C 0.000 }
gfCNCPoint6[9463] = {X 432.5144, Y 49.2400, Z -8.0000, A 0.000, B 0.000, C 0.000 }
gfCNCPoint6[9464] = {X 431.5709, Y 49.1337, Z -8.0000, A 0.000, B 0.000, C 0.000 }
gfCNCPoint6[9465] = {X 430.6748, Y 48.8201, Z -8.0000, A 0.000, B 0.000, C 0.000 }
gfCNCPoint6[9466] = {X 429.8708, Y 48.3150, Z -8.0000, A 0.000, B 0.000, C 0.000 }
gfCNCPoint6[9467] = {X 429.1995, Y 47.6436, Z -8.0000, A 0.000, B 0.000, C 0.000 }
gfCNCPoint6[9468] = {X 428.6943, Y 46.8397, Z -8.0000, A 0.000, B 0.000, C 0.000 }
gfCNCPoint6[9469] = {X 428.3807, Y 45.9436, Z -8.0000, A 0.000, B 0.000, C 0.000 }
gfCNCPoint6[9470] = {X 428.2744, Y 45.0001, Z -8.0000, A 0.000, B 0.000, C 0.000 }
gfCNCPoint6[9471] = {X 428.2748, Y 44.1505, Z -8.0000, A 0.000, B 0.000, C 0.000 }
gfCNCPoint6[9472] = {X 428.3718, Y 43.3054, Z -8.0000, A 0.000, B 0.000, C 0.000 }
gfCNCPoint6[9473] = {X 428.6354, Y 42.4967, Z -8.0000, A 0.000, B 0.000, C 0.000 }
gfCNCPoint6[9474] = {X 429.0552, Y 41.7570, Z -8.0000, A 0.000, B 0.000, C 0.000 }
gfCNCPoint6[9475] = {X 429.6142, Y 41.1158, Z -8.0000, A 0.000, B 0.000, C 0.000 }
gfCNCPoint6[9476] = {X 430.2899, Y 40.5992, Z -8.0000, A 0.000, B 0.000, C 0.000 }
gfCNCPoint6[9477] = {X 431.0551, Y 40.2278, Z -8.0000, A 0.000, B 0.000, C 0.000 }
gfCNCPoint6[9478] = {X 435.0924, Y 32.3253, Z -8.0000, A 0.000, B 0.000, C 0.000 }
gfCNCPoint6[9479] = {X 433.9217, Y 31.5490, Z -8.0000, A 0.000, B 0.000, C 0.000 }
gfCNCPoint6[9480] = {X 432.8568, Y 30.6330, Z -8.0000, A 0.000, B 0.000, C 0.000 }
gfCNCPoint6[9481] = {X 431.9144, Y 29.5914, Z -8.0000, A 0.000, B 0.000, C 0.000 }
gfCNCPoint6[9482] = {X 431.1090, Y 28.4405, Z -8.0000, A 0.000, B 0.000, C 0.000 }
gfCNCPoint6[9483] = {X 430.4534, Y 27.1982, Z -8.0000, A 0.000, B 0.000, C 0.000 }
gfCNCPoint6[9484] = {X 429.9576, Y 25.8839, Z -8.0000, A 0.000, B 0.000, C 0.000 }
gfCNCPoint6[9485] = {X 429.5282, Y 24.0465, Z -8.0000, A 0.000, B 0.000, C 0.000 }
gfCNCPoint6[9486] = {X 429.3120, Y 22.1721, Z -8.0000, A 0.000, B 0.000, C 0.000 }
gfCNCPoint6[9487] = {X 429.3118, Y 20.2852, Z -8.0000, A 0.000, B 0.000, C 0.000 }
gfCNCPoint6[9488] = {X 429.5277, Y 18.4106, Z -8.0000, A 0.000, B 0.000, C 0.000 }
gfCNCPoint6[9489] = {X 429.9568, Y 16.5732, Z -8.0000, A 0.000, B 0.000, C 0.000 }
gfCNCPoint6[9490] = {X 430.5227, Y 15.0523, Z -8.0000, A 0.000, B 0.000, C 0.000 }
gfCNCPoint6[9491] = {X 431.2928, Y 13.6240, Z -8.0000, A 0.000, B 0.000, C 0.000 }
gfCNCPoint6[9492] = {X 432.2524, Y 12.3153, Z -8.0000, A 0.000, B 0.000, C 0.000 }
gfCNCPoint6[9493] = {X 433.3830, Y 11.1513, Z -8.0000, A 0.000, B 0.000, C 0.000 }
gfCNCPoint6[9494] = {X 434.6633, Y 10.1543, Z -8.0000, A 0.000, B 0.000, C 0.000 }
gfCNCPoint6[9495] = {X 436.0688, Y 9.3431, Z -8.0000, A 0.000, B 0.000, C 0.000 }
gfCNCPoint6[9496] = {X 437.5726, Y 8.7333, Z -8.0000, A 0.000, B 0.000, C 0.000 }
gfCNCPoint6[9497] = {X 439.1460, Y 8.3365, Z -8.0000, A 0.000, B 0.000, C 0.000 }
gfCNCPoint6[9498] = {X 441.2360, Y 8.0472, Z -8.0000, A 0.000, B 0.000, C 0.000 }
gfCNCPoint6[9499] = {X 443.3437, Y 7.9533, Z -8.0000, A 0.000, B 0.000, C 0.000 }
gfCNCPoint6[9500] = {X 444.0360, Y 7.9492, Z -8.0000, A 0.000, B 0.000, C 0.000 }
gfCNCPoint6[9501] = {X 459.4469, Y 7.9492, Z -8.0000, A 0.000, B 0.000, C 0.000 }
gfCNCPoint6[9502] = {X 460.3884, Y 8.0553, Z -8.0000, A 0.000, B 0.000, C 0.000 }
gfCNCPoint6[9503] = {X 461.2827, Y 8.3682, Z -8.0000, A 0.000, B 0.000, C 0.000 }
gfCNCPoint6[9504] = {X 462.0849, Y 8.8723, Z -8.0000, A 0.000, B 0.000, C 0.000 }
gfCNCPoint6[9505] = {X 462.7549, Y 9.5423, Z -8.0000, A 0.000, B 0.000, C 0.000 }
gfCNCPoint6[9506] = {X 463.2589, Y 10.3445, Z -8.0000, A 0.000, B 0.000, C 0.000 }
gfCNCPoint6[9507] = {X 463.5719, Y 11.2388, Z -8.0000, A 0.000, B 0.000, C 0.000 }
gfCNCPoint6[9508] = {X 463.6779, Y 12.1803, Z -8.0000, A 0.000, B 0.000, C 0.000 }
gfCNCPoint6[9509] = {X 463.6779, Y 12.9782, Z -8.0000, A 0.000, B 0.000, C 0.000 }
gfCNCPoint6[9510] = {X 463.5765, Y 13.8994, Z -8.0000, A 0.000, B 0.000, C 0.000 }
gfCNCPoint6[9511] = {X 463.2774, Y 14.7766, Z -8.0000, A 0.000, B 0.000, C 0.000 }
gfCNCPoint6[9512] = {X 462.7948, Y 15.5678, Z -8.0000, A 0.000, B 0.000, C 0.000 }
gfCNCPoint6[9513] = {X 462.1518, Y 16.2353, Z -8.0000, A 0.000, B 0.000, C 0.000 }
gfCNCPoint6[9514] = {X 462.1520, Y 28.5935, Z -8.0000, A 0.000, B 0.000, C 0.000 }
gfCNCPoint6[9515] = {X 466.1520, Y 28.5934, Z -8.0000, A 0.000, B 0.000, C 0.000 }
gfCNCPoint6[9516] = {X 462.0720, Y 28.5935, Z -8.0000, A 0.000, B 0.000, C 0.000 }
gfCNCPoint6[9517] = {X 462.0723, Y 40.9896, Z -8.0000, A 0.000, B 0.000, C 0.000 }
gfCNCPoint6[9518] = {X 462.1376, Y 41.0437, Z -8.0000, A 0.000, B 0.000, C 0.000 }
gfCNCPoint6[9519] = {X 462.7482, Y 41.6893, Z -8.0000, A 0.000, B 0.000, C 0.000 }
gfCNCPoint6[9520] = {X 463.2077, Y 42.4498, Z -8.0000, A 0.000, B 0.000, C 0.000 }
gfCNCPoint6[9521] = {X 463.4953, Y 43.2905, Z -8.0000, A 0.000, B 0.000, C 0.000 }
gfCNCPoint6[9522] = {X 463.5978, Y 44.1731, Z -8.0000, A 0.000, B 0.000, C 0.000 }
gfCNCPoint6[9523] = {X 463.5979, Y 45.0000, Z -8.0000, A 0.000, B 0.000, C 0.000 }
gfCNCPoint6[9524] = {X 463.4936, Y 45.9257, Z -8.0000, A 0.000, B 0.000, C 0.000 }
gfCNCPoint6[9525] = {X 463.1860, Y 46.8050, Z -8.0000, A 0.000, B 0.000, C 0.000 }
gfCNCPoint6[9526] = {X 462.6904, Y 47.5937, Z -8.0000, A 0.000, B 0.000, C 0.000 }
gfCNCPoint6[9527] = {X 462.0317, Y 48.2524, Z -8.0000, A 0.000, B 0.000, C 0.000 }
gfCNCPoint6[9528] = {X 461.2429, Y 48.7480, Z -8.0000, A 0.000, B 0.000, C 0.000 }
gfCNCPoint6[9529] = {X 460.3636, Y 49.0557, Z -8.0000, A 0.000, B 0.000, C 0.000 }
gfCNCPoint6[9530] = {X 459.4379, Y 49.1600, Z -8.0000, A 0.000, B 0.000, C 0.000 }
gfCNCPoint6[9531] = {X 452.9945, Y 49.1600, Z -8.0000, A 0.000, B 0.000, C 0.000 }
gfCNCPoint6[9532] = {X 452.0735, Y 49.0568, Z -8.0000, A 0.000, B 0.000, C 0.000 }
gfCNCPoint6[9533] = {X 451.1982, Y 48.7522, Z -8.0000, A 0.000, B 0.000, C 0.000 }
gfCNCPoint6[9534] = {X 450.4120, Y 48.2614, Z -8.0000, A 0.000, B 0.000, C 0.000 }
gfCNCPoint6[9535] = {X 449.7541, Y 47.6087, Z -8.0000, A 0.000, B 0.000, C 0.000 }
gfCNCPoint6[9536] = {X 449.2569, Y 46.8266, Z -8.0000, A 0.000, B 0.000, C 0.000 }
gfCNCPoint6[9537] = {X 448.9453, Y 45.9538, Z -8.0000, A 0.000, B 0.000, C 0.000 }
gfCNCPoint6[9538] = {X 448.8346, Y 45.0336, Z -8.0000, A 0.000, B 0.000, C 0.000 }
gfCNCPoint6[9539] = {X 448.8349, Y 44.1516, Z -8.0000, A 0.000, B 0.000, C 0.000 }
gfCNCPoint6[9540] = {X 448.9454, Y 43.2545, Z -8.0000, A 0.000, B 0.000, C 0.000 }
gfCNCPoint6[9541] = {X 449.2471, Y 42.4026, Z -8.0000, A 0.000, B 0.000, C 0.000 }
gfCNCPoint6[9542] = {X 449.7256, Y 41.6358, Z -8.0000, A 0.000, B 0.000, C 0.000 }
gfCNCPoint6[9543] = {X 450.3584, Y 40.9906, Z -8.0000, A 0.000, B 0.000, C 0.000 }
gfCNCPoint6[9544] = {X 450.3584, Y 34.3138, Z -8.0000, A 0.000, B 0.000, C 0.000 }
gfCNCPoint6[9545] = {X 447.3780, Y 34.3138, Z -8.0000, A 0.000, B 0.000, C 0.000 }
gfCNCPoint6[9546] = {X 443.0163, Y 42.8067, Z -8.0000, A 0.000, B 0.000, C 0.000 }
gfCNCPoint6[9547] = {X 443.0439, Y 42.8839, Z -8.0000, A 0.000, B 0.000, C 0.000 }
gfCNCPoint6[9548] = {X 443.2029, Y 43.5193, Z -8.0000, A 0.000, B 0.000, C 0.000 }
gfCNCPoint6[9549] = {X 443.2603, Y 44.1717, Z -8.0000, A 0.000, B 0.000, C 0.000 }
gfCNCPoint6[9550] = {X 443.2605, Y 45.0000, Z -8.0000, A 0.000, B 0.000, C 0.000 }
gfCNCPoint6[9551] = {X 443.1562, Y 45.9257, Z -8.0000, A 0.000, B 0.000, C 0.000 }
gfCNCPoint6[9552] = {X 442.8485, Y 46.8050, Z -8.0000, A 0.000, B 0.000, C 0.000 }
gfCNCPoint6[9553] = {X 442.3529, Y 47.5937, Z -8.0000, A 0.000, B 0.000, C 0.000 }
gfCNCPoint6[9554] = {X 441.6942, Y 48.2524, Z -8.0000, A 0.000, B 0.000, C 0.000 }
gfCNCPoint6[9555] = {X 440.9054, Y 48.7480, Z -8.0000, A 0.000, B 0.000, C 0.000 }
gfCNCPoint6[9556] = {X 440.0262, Y 49.0557, Z -8.0000, A 0.000, B 0.000, C 0.000 }
gfCNCPoint6[9557] = {X 439.1005, Y 49.1600, Z -8.0000, A 0.000, B 0.000, C 0.000 }
gfCNCPoint6[9558] = {X 432.5144, Y 49.1600, Z -8.0000, A 0.000, B 0.000, C 0.000 }
gfCNCPoint6[9559] = {X 431.5887, Y 49.0557, Z -8.0000, A 0.000, B 0.000, C 0.000 }
gfCNCPoint6[9560] = {X 430.7095, Y 48.7480, Z -8.0000, A 0.000, B 0.000, C 0.000 }
gfCNCPoint6[9561] = {X 429.9207, Y 48.2524, Z -8.0000, A 0.000, B 0.000, C 0.000 }
gfCNCPoint6[9562] = {X 429.2620, Y 47.5937, Z -8.0000, A 0.000, B 0.000, C 0.000 }
gfCNCPoint6[9563] = {X 428.7664, Y 46.8050, Z -8.0000, A 0.000, B 0.000, C 0.000 }
gfCNCPoint6[9564] = {X 428.4587, Y 45.9257, Z -8.0000, A 0.000, B 0.000, C 0.000 }
gfCNCPoint6[9565] = {X 428.3544, Y 45.0000, Z -8.0000, A 0.000, B 0.000, C 0.000 }
gfCNCPoint6[9566] = {X 428.3548, Y 44.1516, Z -8.0000, A 0.000, B 0.000, C 0.000 }
gfCNCPoint6[9567] = {X 428.4510, Y 43.3174, Z -8.0000, A 0.000, B 0.000, C 0.000 }
gfCNCPoint6[9568] = {X 428.7128, Y 42.5195, Z -8.0000, A 0.000, B 0.000, C 0.000 }
gfCNCPoint6[9569] = {X 429.1295, Y 41.7905, Z -8.0000, A 0.000, B 0.000, C 0.000 }
gfCNCPoint6[9570] = {X 429.6841, Y 41.1600, Z -8.0000, A 0.000, B 0.000, C 0.000 }
gfCNCPoint6[9571] = {X 430.3541, Y 40.6537, Z -8.0000, A 0.000, B 0.000, C 0.000 }
gfCNCPoint6[9572] = {X 431.1120, Y 40.2923, Z -8.0000, A 0.000, B 0.000, C 0.000 }
gfCNCPoint6[9573] = {X 435.1983, Y 32.2938, Z -8.0000, A 0.000, B 0.000, C 0.000 }
gfCNCPoint6[9574] = {X 434.0206, Y 31.5234, Z -8.0000, A 0.000, B 0.000, C 0.000 }
gfCNCPoint6[9575] = {X 432.9490, Y 30.6110, Z -8.0000, A 0.000, B 0.000, C 0.000 }
gfCNCPoint6[9576] = {X 432.0007, Y 29.5712, Z -8.0000, A 0.000, B 0.000, C 0.000 }
gfCNCPoint6[9577] = {X 431.1905, Y 28.4204, Z -8.0000, A 0.000, B 0.000, C 0.000 }
gfCNCPoint6[9578] = {X 430.5315, Y 27.1769, Z -8.0000, A 0.000, B 0.000, C 0.000 }
gfCNCPoint6[9579] = {X 430.0341, Y 25.8604, Z -8.0000, A 0.000, B 0.000, C 0.000 }
gfCNCPoint6[9580] = {X 429.6069, Y 24.0321, Z -8.0000, A 0.000, B 0.000, C 0.000 }
gfCNCPoint6[9581] = {X 429.3918, Y 22.1669, Z -8.0000, A 0.000, B 0.000, C 0.000 }
gfCNCPoint6[9582] = {X 429.3917, Y 20.2894, Z -8.0000, A 0.000, B 0.000, C 0.000 }
gfCNCPoint6[9583] = {X 429.6066, Y 18.4242, Z -8.0000, A 0.000, B 0.000, C 0.000 }
gfCNCPoint6[9584] = {X 430.0335, Y 16.5958, Z -8.0000, A 0.000, B 0.000, C 0.000 }
gfCNCPoint6[9585] = {X 430.5956, Y 15.0853, Z -8.0000, A 0.000, B 0.000, C 0.000 }
gfCNCPoint6[9586] = {X 431.3605, Y 13.6666, Z -8.0000, A 0.000, B 0.000, C 0.000 }
gfCNCPoint6[9587] = {X 432.3135, Y 12.3669, Z -8.0000, A 0.000, B 0.000, C 0.000 }
gfCNCPoint6[9588] = {X 433.4365, Y 11.2108, Z -8.0000, A 0.000, B 0.000, C 0.000 }
gfCNCPoint6[9589] = {X 434.7081, Y 10.2205, Z -8.0000, A 0.000, B 0.000, C 0.000 }
gfCNCPoint6[9590] = {X 436.1041, Y 9.4149, Z -8.0000, A 0.000, B 0.000, C 0.000 }
gfCNCPoint6[9591] = {X 437.5977, Y 8.8093, Z -8.0000, A 0.000, B 0.000, C 0.000 }
gfCNCPoint6[9592] = {X 439.1605, Y 8.4152, Z -8.0000, A 0.000, B 0.000, C 0.000 }
gfCNCPoint6[9593] = {X 441.2433, Y 8.1268, Z -8.0000, A 0.000, B 0.000, C 0.000 }
gfCNCPoint6[9594] = {X 443.3439, Y 8.0333, Z -8.0000, A 0.000, B 0.000, C 0.000 }
gfCNCPoint6[9595] = {X 444.0362, Y 8.0292, Z -8.0000, A 0.000, B 0.000, C 0.000 }
gfCNCPoint6[9596] = {X 459.4469, Y 8.0292, Z -8.0000, A 0.000, B 0.000, C 0.000 }
gfCNCPoint6[9597] = {X 460.3706, Y 8.1333, Z -8.0000, A 0.000, B 0.000, C 0.000 }
gfCNCPoint6[9598] = {X 461.2480, Y 8.4403, Z -8.0000, A 0.000, B 0.000, C 0.000 }
gfCNCPoint6[9599] = {X 462.0350, Y 8.9349, Z -8.0000, A 0.000, B 0.000, C 0.000 }
gfCNCPoint6[9600] = {X 462.6923, Y 9.5921, Z -8.0000, A 0.000, B 0.000, C 0.000 }
gfCNCPoint6[9601] = {X 463.1869, Y 10.3792, Z -8.0000, A 0.000, B 0.000, C 0.000 }
gfCNCPoint6[9602] = {X 463.4939, Y 11.2566, Z -8.0000, A 0.000, B 0.000, C 0.000 }
gfCNCPoint6[9603] = {X 463.5979, Y 12.1803, Z -8.0000, A 0.000, B 0.000, C 0.000 }
gfCNCPoint6[9604] = {X 463.5979, Y 12.9782, Z -8.0000, A 0.000, B 0.000, C 0.000 }
gfCNCPoint6[9605] = {X 463.5023, Y 13.8647, Z -8.0000, A 0.000, B 0.000, C 0.000 }
gfCNCPoint6[9606] = {X 463.2200, Y 14.7105, Z -8.0000, A 0.000, B 0.000, C 0.000 }
gfCNCPoint6[9607] = {X 462.7639, Y 15.4767, Z -8.0000, A 0.000, B 0.000, C 0.000 }
gfCNCPoint6[9608] = {X 462.1550, Y 16.1282, Z -8.0000, A 0.000, B 0.000, C 0.000 }
gfCNCPoint6[9609] = {X 462.0718, Y 16.1980, Z -8.0000, A 0.000, B 0.000, C 0.000 }
gfCNCPoint6[9610] = {X 462.0720, Y 28.5935, Z -8.0000, A 0.000, B 0.000, C 0.000 }
gfCNCPoint6[9611] = {X 466.0720, Y 28.5934, Z -8.0000, A 0.000, B 0.000, C 0.000 }
gfCNCPoint6[9612] = {X 461.9920, Y 28.5935, Z -8.0000, A 0.000, B 0.000, C 0.000 }
gfCNCPoint6[9613] = {X 461.9923, Y 41.0272, Z -8.0000, A 0.000, B 0.000, C 0.000 }
gfCNCPoint6[9614] = {X 462.0861, Y 41.1050, Z -8.0000, A 0.000, B 0.000, C 0.000 }
gfCNCPoint6[9615] = {X 462.6848, Y 41.7381, Z -8.0000, A 0.000, B 0.000, C 0.000 }
gfCNCPoint6[9616] = {X 463.1354, Y 42.4838, Z -8.0000, A 0.000, B 0.000, C 0.000 }
gfCNCPoint6[9617] = {X 463.4173, Y 43.3083, Z -8.0000, A 0.000, B 0.000, C 0.000 }
gfCNCPoint6[9618] = {X 463.5178, Y 44.1738, Z -8.0000, A 0.000, B 0.000, C 0.000 }
gfCNCPoint6[9619] = {X 463.5179, Y 45.0000, Z -8.0000, A 0.000, B 0.000, C 0.000 }
gfCNCPoint6[9620] = {X 463.4156, Y 45.9079, Z -8.0000, A 0.000, B 0.000, C 0.000 }
gfCNCPoint6[9621] = {X 463.1139, Y 46.7702, Z -8.0000, A 0.000, B 0.000, C 0.000 }
gfCNCPoint6[9622] = {X 462.6278, Y 47.5438, Z -8.0000, A 0.000, B 0.000, C 0.000 }
gfCNCPoint6[9623] = {X 461.9818, Y 48.1899, Z -8.0000, A 0.000, B 0.000, C 0.000 }
gfCNCPoint6[9624] = {X 461.2082, Y 48.6760, Z -8.0000, A 0.000, B 0.000, C 0.000 }
gfCNCPoint6[9625] = {X 460.3458, Y 48.9777, Z -8.0000, A 0.000, B 0.000, C 0.000 }
gfCNCPoint6[9626] = {X 459.4379, Y 49.0800, Z -8.0000, A 0.000, B 0.000, C 0.000 }
gfCNCPoint6[9627] = {X 452.9945, Y 49.0800, Z -8.0000, A 0.000, B 0.000, C 0.000 }
gfCNCPoint6[9628] = {X 452.0912, Y 48.9788, Z -8.0000, A 0.000, B 0.000, C 0.000 }
gfCNCPoint6[9629] = {X 451.2327, Y 48.6800, Z -8.0000, A 0.000, B 0.000, C 0.000 }
gfCNCPoint6[9630] = {X 450.4617, Y 48.1987, Z -8.0000, A 0.000, B 0.000, C 0.000 }
gfCNCPoint6[9631] = {X 449.8164, Y 47.5585, Z -8.0000, A 0.000, B 0.000, C 0.000 }
gfCNCPoint6[9632] = {X 449.3288, Y 46.7914, Z -8.0000, A 0.000, B 0.000, C 0.000 }
gfCNCPoint6[9633] = {X 449.0232, Y 45.9354, Z -8.0000, A 0.000, B 0.000, C 0.000 }
gfCNCPoint6[9634] = {X 448.9146, Y 45.0330, Z -8.0000, A 0.000, B 0.000, C 0.000 }
gfCNCPoint6[9635] = {X 448.9149, Y 44.1527, Z -8.0000, A 0.000, B 0.000, C 0.000 }
gfCNCPoint6[9636] = {X 449.0254, Y 43.2637, Z -8.0000, A 0.000, B 0.000, C 0.000 }
gfCNCPoint6[9637] = {X 449.3274, Y 42.4203, Z -8.0000, A 0.000, B 0.000, C 0.000 }
gfCNCPoint6[9638] = {X 449.8061, Y 41.6631, Z -8.0000, A 0.000, B 0.000, C 0.000 }
gfCNCPoint6[9639] = {X 450.4384, Y 41.0287, Z -8.0000, A 0.000, B 0.000, C 0.000 }
gfCNCPoint6[9640] = {X 450.4384, Y 34.2338, Z -8.0000, A 0.000, B 0.000, C 0.000 }
gfCNCPoint6[9641] = {X 447.3291, Y 34.2338, Z -8.0000, A 0.000, B 0.000, C 0.000 }
gfCNCPoint6[9642] = {X 442.9293, Y 42.8010, Z -8.0000, A 0.000, B 0.000, C 0.000 }
gfCNCPoint6[9643] = {X 442.9683, Y 42.9101, Z -8.0000, A 0.000, B 0.000, C 0.000 }
gfCNCPoint6[9644] = {X 443.1241, Y 43.5329, Z -8.0000, A 0.000, B 0.000, C 0.000 }
gfCNCPoint6[9645] = {X 443.1803, Y 44.1725, Z -8.0000, A 0.000, B 0.000, C 0.000 }
gfCNCPoint6[9646] = {X 443.1805, Y 45.0000, Z -8.0000, A 0.000, B 0.000, C 0.000 }
gfCNCPoint6[9647] = {X 443.0782, Y 45.9079, Z -8.0000, A 0.000, B 0.000, C 0.000 }
gfCNCPoint6[9648] = {X 442.7764, Y 46.7702, Z -8.0000, A 0.000, B 0.000, C 0.000 }
gfCNCPoint6[9649] = {X 442.2903, Y 47.5438, Z -8.0000, A 0.000, B 0.000, C 0.000 }
gfCNCPoint6[9650] = {X 441.6443, Y 48.1899, Z -8.0000, A 0.000, B 0.000, C 0.000 }
gfCNCPoint6[9651] = {X 440.8707, Y 48.6760, Z -8.0000, A 0.000, B 0.000, C 0.000 }
gfCNCPoint6[9652] = {X 440.0084, Y 48.9777, Z -8.0000, A 0.000, B 0.000, C 0.000 }
gfCNCPoint6[9653] = {X 439.1005, Y 49.0800, Z -8.0000, A 0.000, B 0.000, C 0.000 }
gfCNCPoint6[9654] = {X 432.5144, Y 49.0800, Z -8.0000, A 0.000, B 0.000, C 0.000 }
gfCNCPoint6[9655] = {X 431.6065, Y 48.9777, Z -8.0000, A 0.000, B 0.000, C 0.000 }
gfCNCPoint6[9656] = {X 430.7442, Y 48.6760, Z -8.0000, A 0.000, B 0.000, C 0.000 }
gfCNCPoint6[9657] = {X 429.9706, Y 48.1899, Z -8.0000, A 0.000, B 0.000, C 0.000 }
gfCNCPoint6[9658] = {X 429.3245, Y 47.5438, Z -8.0000, A 0.000, B 0.000, C 0.000 }
gfCNCPoint6[9659] = {X 428.8385, Y 46.7702, Z -8.0000, A 0.000, B 0.000, C 0.000 }
gfCNCPoint6[9660] = {X 428.5367, Y 45.9079, Z -8.0000, A 0.000, B 0.000, C 0.000 }
gfCNCPoint6[9661] = {X 428.4344, Y 45.0000, Z -8.0000, A 0.000, B 0.000, C 0.000 }
gfCNCPoint6[9662] = {X 428.4348, Y 44.1527, Z -8.0000, A 0.000, B 0.000, C 0.000 }
gfCNCPoint6[9663] = {X 428.5303, Y 43.3294, Z -8.0000, A 0.000, B 0.000, C 0.000 }
gfCNCPoint6[9664] = {X 428.7902, Y 42.5424, Z -8.0000, A 0.000, B 0.000, C 0.000 }
gfCNCPoint6[9665] = {X 429.2038, Y 41.8242, Z -8.0000, A 0.000, B 0.000, C 0.000 }
gfCNCPoint6[9666] = {X 429.7540, Y 41.2044, Z -8.0000, A 0.000, B 0.000, C 0.000 }
gfCNCPoint6[9667] = {X 430.4181, Y 40.7085, Z -8.0000, A 0.000, B 0.000, C 0.000 }
gfCNCPoint6[9668] = {X 431.1687, Y 40.3571, Z -8.0000, A 0.000, B 0.000, C 0.000 }
gfCNCPoint6[9669] = {X 435.3045, Y 32.2617, Z -8.0000, A 0.000, B 0.000, C 0.000 }
gfCNCPoint6[9670] = {X 434.1197, Y 31.4974, Z -8.0000, A 0.000, B 0.000, C 0.000 }
gfCNCPoint6[9671] = {X 433.0414, Y 30.5889, Z -8.0000, A 0.000, B 0.000, C 0.000 }
gfCNCPoint6[9672] = {X 432.0871, Y 29.5509, Z -8.0000, A 0.000, B 0.000, C 0.000 }
gfCNCPoint6[9673] = {X 431.2721, Y 28.4003, Z -8.0000, A 0.000, B 0.000, C 0.000 }
gfCNCPoint6[9674] = {X 430.6097, Y 27.1556, Z -8.0000, A 0.000, B 0.000, C 0.000 }
gfCNCPoint6[9675] = {X 430.1105, Y 25.8369, Z -8.0000, A 0.000, B 0.000, C 0.000 }
gfCNCPoint6[9676] = {X 429.6856, Y 24.0177, Z -8.0000, A 0.000, B 0.000, C 0.000 }
gfCNCPoint6[9677] = {X 429.4717, Y 22.1618, Z -8.0000, A 0.000, B 0.000, C 0.000 }
gfCNCPoint6[9678] = {X 429.4716, Y 20.2936, Z -8.0000, A 0.000, B 0.000, C 0.000 }
